# B&R Automation Studio project CombinedLinenCleanA6 (part 6)

```automation-basic
	; ###HO - 260905 - a_usCustomize[0..6]
		if(TARGETInfo_0.DataFormat = 2) then  ; motorola
			memcpy(adr(LocalCAN2Data.T3_By1),adr(LocalCOB_Typ_307.a_usCustomize[0]),1)
			memcpy(adr(LocalCAN2Data.T3_By2_By3),adr(LocalCOB_Typ_307.a_usCustomize[1]),2)
			memcpy(adr(LocalCAN2Data.T3_By4_By5),adr(LocalCOB_Typ_307.a_usCustomize[3]),2)
			memcpy(adr(LocalCAN2Data.T3_By6_By7),adr(LocalCOB_Typ_307.a_usCustomize[5]),2)
		else ; intel
			LocalCAN2Data.T3_By1 	 = LocalCOB_Typ_307.a_usCustomize[0]
			LocalCAN2Data.T3_By2_By3 = LocalCOB_Typ_307.a_usCustomize[2] + 256* LocalCOB_Typ_307.a_usCustomize[1]
			LocalCAN2Data.T3_By4_By5 = LocalCOB_Typ_307.a_usCustomize[4] + 256* LocalCOB_Typ_307.a_usCustomize[3]
			LocalCAN2Data.T3_By6_By7 = LocalCOB_Typ_307.a_usCustomize[6] + 256* LocalCOB_Typ_307.a_usCustomize[5]
		endif

    iStatus = 0
    pCAN2Data = ADR(LocalCAN2Data)
endaction ; 307

;*******action 311********action 311********action 311********action 311********action 311********
action 311: ; 311:
action 312: ; 312:
action 313: ; 313:
action 314: ; 314:
    	; ocalCOB_Typ_311 access Local_InitCAN2PV.pPVData
    	memcpy(adr(LocalCOB_Typ_311),Local_InitCAN2PV.pPVData,sizeof(LocalCOB_Typ_311))
;****ID 311****Telegram 1********ID 311****Telegram 1********ID 311****Telegram 1********ID 311****Telegram 1****
	;T1 mandatotries ->:
	; .. and sign CAN2 telegram
	LocalCAN2Data.T1_By0 = BIT_CLR(LocalCAN2Data.T1_By0, 6)
	LocalCAN2Data.T1_By0 = BIT_SET(LocalCAN2Data.T1_By0, 7)

		; bBereit
    	if LocalCOB_Typ_311.bBereit = 1 then
			LocalCAN2Data.T1_By0 = BIT_SET(LocalCAN2Data.T1_By0, 0)
		else
			LocalCAN2Data.T1_By0 = BIT_CLR(LocalCAN2Data.T1_By0, 0)
		endif
		; bBeladebereit
    	if LocalCOB_Typ_311.bBeladebereit = 1 then
			LocalCAN2Data.T1_By0 = BIT_SET(LocalCAN2Data.T1_By0, 1)
		else
			LocalCAN2Data.T1_By0 = BIT_CLR(LocalCAN2Data.T1_By0, 1)
		endif
		; bStartPresse
    	if LocalCOB_Typ_311.bStartPresse = 1 then
			LocalCAN2Data.T1_By0 = BIT_SET(LocalCAN2Data.T1_By0, 2)
		else
			LocalCAN2Data.T1_By0 = BIT_CLR(LocalCAN2Data.T1_By0, 2)
		endif
		; bUebernahmestoerungVerbETAero
    	if LocalCOB_Typ_311.bUebernahmestoerungVerbETAero = 1 then
			LocalCAN2Data.T1_By0 = BIT_SET(LocalCAN2Data.T1_By0, 3)
		else
			LocalCAN2Data.T1_By0 = BIT_CLR(LocalCAN2Data.T1_By0, 3)
		endif
		; bEntladelichtschrZentrifuge
    	if LocalCOB_Typ_311.bEntladelichtschrZentrifuge	 = 1 then
			LocalCAN2Data.T1_By0 = BIT_SET(LocalCAN2Data.T1_By0, 4)
		else
			LocalCAN2Data.T1_By0 = BIT_CLR(LocalCAN2Data.T1_By0, 4)
		endif
   ; bNotAusETVerbAero
	    if LocalCOB_Typ_311.bNotAusETVerbAero = 1 then
			LocalCAN2Data.T1_By1 = BIT_SET(LocalCAN2Data.T1_By1, 0)
		else
			LocalCAN2Data.T1_By1 = BIT_CLR(LocalCAN2Data.T1_By1, 0)
		endif
   ; bSchutzgitterOffen
	    if LocalCOB_Typ_311.bSchutzgitterOffen = 1 then
			LocalCAN2Data.T1_By1 = BIT_SET(LocalCAN2Data.T1_By1, 1)
		else
			LocalCAN2Data.T1_By1 = BIT_CLR(LocalCAN2Data.T1_By1, 1)
		endif

;****ID 311****Telegram 2********ID 311****Telegram 2********ID 311****Telegram 2********ID 311****Telegram 2****
	;T1 mandatotries ->:
	; .. and sign CAN2 telegram
	LocalCAN2Data.T2_By0 = BIT_SET(LocalCAN2Data.T2_By0, 6)
	LocalCAN2Data.T2_By0 = BIT_SET(LocalCAN2Data.T2_By0, 7)

	; ###HO - 230905 - a_usCustomize[0..6]
		if(TARGETInfo_0.DataFormat = 2) then  ; motorola
			memcpy(adr(LocalCAN2Data.T2_By1),adr(LocalCOB_Typ_311.a_usCustomize[0]),1)
			memcpy(adr(LocalCAN2Data.T2_By2_By3),adr(LocalCOB_Typ_311.a_usCustomize[1]),2)
			memcpy(adr(LocalCAN2Data.T2_By4_By5),adr(LocalCOB_Typ_311.a_usCustomize[3]),2)
			memcpy(adr(LocalCAN2Data.T2_By6_By7),adr(LocalCOB_Typ_311.a_usCustomize[5]),2)
		else ; intel
			LocalCAN2Data.T2_By1 	 = LocalCOB_Typ_311.a_usCustomize[0]
			LocalCAN2Data.T2_By2_By3 = LocalCOB_Typ_311.a_usCustomize[2] + 256* LocalCOB_Typ_311.a_usCustomize[1]
			LocalCAN2Data.T2_By4_By5 = LocalCOB_Typ_311.a_usCustomize[4] + 256* LocalCOB_Typ_311.a_usCustomize[3]
			LocalCAN2Data.T2_By6_By7 = LocalCOB_Typ_311.a_usCustomize[6] + 256* LocalCOB_Typ_311.a_usCustomize[5]
		endif

        iStatus = 0
        pCAN2Data = ADR(LocalCAN2Data)
endaction ; 311
;-----------------------------------------------------------------------------------------------------------------

;-----------------------------------------------------------------------------------------------------------------

action 316:	; 316:
    ; pLocalCOB_Typ_316 access Local_InitCAN2PV.pPVData
    memcpy(adr(LocalCOB_Typ_316),Local_InitCAN2PV.pPVData,sizeof(LocalCOB_Typ_316))
;****ID 316****Telegram 1********ID 316****Telegram 1********ID 316****Telegram 1********ID 316****Telegram 1****
	;T1 mandatotries ->:
	LocalCAN2Data.T1_By0 = BIT_CLR(LocalCAN2Data.T1_By0, 5)
	LocalCAN2Data.T1_By0 = BIT_CLR(LocalCAN2Data.T1_By0, 6)
	; .. and sign CAN2 telegram
	LocalCAN2Data.T1_By0 = BIT_SET(LocalCAN2Data.T1_By0, 7)

	; bNotAusVerbET
	   	if LocalCOB_Typ_316.bNotAusVerbET = 1 then
			LocalCAN2Data.T1_By0 = BIT_SET(LocalCAN2Data.T1_By0, 4)
		else
			LocalCAN2Data.T1_By0 = BIT_CLR(LocalCAN2Data.T1_By0, 4)
		endif
	; bBereit
    	if LocalCOB_Typ_316.bBereit = 1 then
			LocalCAN2Data.T1_By0 = BIT_SET(LocalCAN2Data.T1_By0, 0)
		else
			LocalCAN2Data.T1_By0 = BIT_CLR(LocalCAN2Data.T1_By0, 0)
		endif
	; bBeladebereit
    	if LocalCOB_Typ_316.bBeladebereit = 1 then
			LocalCAN2Data.T1_By0 = BIT_SET(LocalCAN2Data.T1_By0, 1)
		else
			LocalCAN2Data.T1_By0 = BIT_CLR(LocalCAN2Data.T1_By0, 1)
		endif
	; bUebernahmestoerungVerbET
    	if LocalCOB_Typ_316.bUebernahmestoerungVerbET = 1 then
			LocalCAN2Data.T1_By0 = BIT_SET(LocalCAN2Data.T1_By0, 3)
		else
			LocalCAN2Data.T1_By0 = BIT_CLR(LocalCAN2Data.T1_By0, 3)
		endif

	;****ID 316****Telegram 2********ID 316****Telegram 2********ID 316****Telegram 2********ID 316****Telegram 2****
	;T1 mandatotries ->:
	; .. and sign CAN2 telegram
	LocalCAN2Data.T2_By0 = BIT_SET(LocalCAN2Data.T2_By0, 5)
	LocalCAN2Data.T2_By0 = BIT_CLR(LocalCAN2Data.T2_By0, 6)
	; .. and sign CAN2 telegram
	LocalCAN2Data.T2_By0 = BIT_SET(LocalCAN2Data.T2_By0, 7)

	; ###HO - 230905 - a_usCustomize[0..6]
	if(TARGETInfo_0.DataFormat = 2) then  ; motorola
		memcpy(adr(LocalCAN2Data.T2_By1),adr(LocalCOB_Typ_316.a_usCustomize[0]),1)
		memcpy(adr(LocalCAN2Data.T2_By2_By3),adr(LocalCOB_Typ_316.a_usCustomize[1]),2)
		memcpy(adr(LocalCAN2Data.T2_By4_By5),adr(LocalCOB_Typ_316.a_usCustomize[3]),2)
		memcpy(adr(LocalCAN2Data.T2_By6_By7),adr(LocalCOB_Typ_316.a_usCustomize[5]),2)
	else ; intel
		LocalCAN2Data.T2_By1 	 = LocalCOB_Typ_316.a_usCustomize[0]
		LocalCAN2Data.T2_By2_By3 = LocalCOB_Typ_316.a_usCustomize[2] + 256* LocalCOB_Typ_316.a_usCustomize[1]
		LocalCAN2Data.T2_By4_By5 = LocalCOB_Typ_316.a_usCustomize[4] + 256* LocalCOB_Typ_316.a_usCustomize[3]
		LocalCAN2Data.T2_By6_By7 = LocalCOB_Typ_316.a_usCustomize[6] + 256* LocalCOB_Typ_316.a_usCustomize[5]
	endif

    iStatus = 0
    pCAN2Data = ADR(LocalCAN2Data)

endaction ; 316

;*******action 317********action 317********action 317********action 317********action 317********
action 317: ; 317:
    	; pLocalCOB_Typ_317 access Local_InitCAN2PV.pPVData
    	memcpy(adr(LocalCOB_Typ_317),Local_InitCAN2PV.pPVData,sizeof(LocalCOB_Typ_317))

;****ID 317****Telegram 1********ID 317****Telegram 1********ID 317****Telegram 1********ID 317****Telegram 1****
	;T1 mandatotries ->:
	LocalCAN2Data.T1_By0 = BIT_CLR(LocalCAN2Data.T1_By0, 6)
	; .. and sign CAN2 telegram
	LocalCAN2Data.T1_By0 = BIT_SET(LocalCAN2Data.T1_By0, 7)

;	bBereit
    	if LocalCOB_Typ_317.bBereit = 1 then
			LocalCAN2Data.T1_By0 = BIT_SET(LocalCAN2Data.T1_By0, 0)
		else
			LocalCAN2Data.T1_By0 = BIT_CLR(LocalCAN2Data.T1_By0, 0)
		endif
;	bBeladebereit
    	if LocalCOB_Typ_317.bBeladebereit = 1 then
			LocalCAN2Data.T1_By0 = BIT_SET(LocalCAN2Data.T1_By0, 1)
		else
			LocalCAN2Data.T1_By0 = BIT_CLR(LocalCAN2Data.T1_By0, 1)
		endif
;	bBeladeunterbrechung
    	if LocalCOB_Typ_317.bBeladeunterbrechung = 1 then
			LocalCAN2Data.T1_By0 = BIT_SET(LocalCAN2Data.T1_By0, 2)
		else
			LocalCAN2Data.T1_By0 = BIT_CLR(LocalCAN2Data.T1_By0, 2)
		endif
;	bUebernahmestoerung
    	if LocalCOB_Typ_317.bUebernahmestoerung = 1 then
			LocalCAN2Data.T1_By0 = BIT_SET(LocalCAN2Data.T1_By0, 3)
		else
			LocalCAN2Data.T1_By0 = BIT_CLR(LocalCAN2Data.T1_By0, 3)
		endif
;	bQuittierungKundenwechsel
    	if LocalCOB_Typ_317.bQuittierungKundenwechsel = 1 then
			LocalCAN2Data.T1_By0 = BIT_SET(LocalCAN2Data.T1_By0, 4)
		else
			LocalCAN2Data.T1_By0 = BIT_CLR(LocalCAN2Data.T1_By0, 4)
		endif
;	bNotAusAero
    	if LocalCOB_Typ_317.bNotAusAero = 1 then
			LocalCAN2Data.T1_By0 = BIT_SET(LocalCAN2Data.T1_By0, 5)
		else
			LocalCAN2Data.T1_By0 = BIT_CLR(LocalCAN2Data.T1_By0, 5)
		endif
;****ID 317****Telegram 2********ID 317****Telegram 2********ID 317****Telegram 2********ID 317****Telegram 2****
	; always set telegram number "01"..
	LocalCAN2Data.T2_By0 = BIT_SET(LocalCAN2Data.T2_By0, 6)
	; .. and sign CAN2 telegram
	LocalCAN2Data.T2_By0 = BIT_SET(LocalCAN2Data.T2_By0, 7)

   	; ###HO - 260905 - a_usCustomize[0..6]
		if(TARGETInfo_0.DataFormat = 2) then  ; motorola
			memcpy(adr(LocalCAN2Data.T2_By1),adr(LocalCOB_Typ_317.a_usCustomize[0]),1)
			memcpy(adr(LocalCAN2Data.T2_By2_By3),adr(LocalCOB_Typ_317.a_usCustomize[1]),2)
			memcpy(adr(LocalCAN2Data.T2_By4_By5),adr(LocalCOB_Typ_317.a_usCustomize[3]),2)
			memcpy(adr(LocalCAN2Data.T2_By6_By7),adr(LocalCOB_Typ_317.a_usCustomize[5]),2)
		else ; intel
			LocalCAN2Data.T2_By1	 = LocalCOB_Typ_317.a_usCustomize[0]
			LocalCAN2Data.T2_By2_By3 = LocalCOB_Typ_317.a_usCustomize[2] + 256* LocalCOB_Typ_317.a_usCustomize[1]
			LocalCAN2Data.T2_By4_By5 = LocalCOB_Typ_317.a_usCustomize[4] + 256* LocalCOB_Typ_317.a_usCustomize[3]
			LocalCAN2Data.T2_By6_By7 = LocalCOB_Typ_317.a_usCustomize[6] + 256* LocalCOB_Typ_317.a_usCustomize[5]
		endif

  	iStatus = 0
    pCAN2Data = ADR(LocalCAN2Data)
endaction ; 317

;*******action 351********action 351********action 351********action 351********action 351********
action 351: ; 351:
    	; pLocalCOB_Typ_351 access Local_InitCAN2PV.pPVData
    	memcpy(adr(LocalCOB_Typ_351),Local_InitCAN2PV.pPVData,sizeof(LocalCOB_Typ_351))

;****ID 351****Telegram 1********ID 351****Telegram 1********ID 351****Telegram 1********ID 351****Telegram 1****
		;T1 mandatotries ->:
		LocalCAN2Data.T1_By0 = BIT_CLR(LocalCAN2Data.T1_By0, 5)
		LocalCAN2Data.T1_By0 = BIT_CLR(LocalCAN2Data.T1_By0, 6)
		; .. and sign CAN2 telegram
		LocalCAN2Data.T1_By0 = BIT_SET(LocalCAN2Data.T1_By0, 7)

;	bBereit
    	if LocalCOB_Typ_351.bBereit = 1 then
			LocalCAN2Data.T1_By0 = BIT_SET(LocalCAN2Data.T1_By0, 0)
		else
				LocalCAN2Data.T1_By0 = BIT_CLR(LocalCAN2Data.T1_By0, 0)
		endif
;	bAktPosFehler
    	if LocalCOB_Typ_351.bAktPosFehler = 1 then
			LocalCAN2Data.T1_By0 = BIT_SET(LocalCAN2Data.T1_By0, 1)
		else
			LocalCAN2Data.T1_By0 = BIT_CLR(LocalCAN2Data.T1_By0, 1)
		endif
;	bIdxPostenindex_x - 110107
    	if LocalCOB_Typ_351.bIdxPostenspeicher_1 = 1 then
			LocalCAN2Data.T1_By0 = BIT_SET(LocalCAN2Data.T1_By0, 2)
		else
			LocalCAN2Data.T1_By0 = BIT_CLR(LocalCAN2Data.T1_By0, 2)
		endif
		if LocalCOB_Typ_351.bIdxPostenspeicher_2 = 1 then
			LocalCAN2Data.T1_By0 = BIT_SET(LocalCAN2Data.T1_By0, 3)
		else
			LocalCAN2Data.T1_By0 = BIT_CLR(LocalCAN2Data.T1_By0, 3)
		endif
		if LocalCOB_Typ_351.bIdxPostenspeicher_4 = 1 then
			LocalCAN2Data.T1_By0 = BIT_SET(LocalCAN2Data.T1_By0, 4)
		else
			LocalCAN2Data.T1_By0 = BIT_CLR(LocalCAN2Data.T1_By0, 4)
		endif
;	usAktPos
		LocalCAN2Data.T1_By1	= LocalCOB_Typ_351.usAktPos
;	udPostennummer				8-11
			udShr16 = shr(LocalCOB_Typ_351.udPostennummer,16)
    	LocalCAN2Data.T1_By2_By3	= UINT(udShr16)							; take UPPERBytes ..
    	LocalCAN2Data.T1_By4_By5	= UINT(LocalCOB_Typ_351.udPostennummer)	; take LOWER byte..
;	uiGewicht					16-17
		LocalCAN2Data.T1_By6_By7	= LocalCOB_Typ_351.uiGewicht

;****ID 351****Telegram 2********ID 351****Telegram 2********ID 351****Telegram 2********ID 351****Telegram 2****
		; always set telegram number "01"..
		LocalCAN2Data.T2_By0 = BIT_CLR(LocalCAN2Data.T2_By0, 5)
		LocalCAN2Data.T2_By0 = BIT_SET(LocalCAN2Data.T2_By0, 6)
		; .. and sign CAN2 telegram
		LocalCAN2Data.T2_By0 = BIT_SET(LocalCAN2Data.T2_By0, 7)

		; bProgrammOderKategorie
    	if LocalCOB_Typ_351.bProgrammOderKategorie = 1 then
			LocalCAN2Data.T2_By0 = BIT_SET(LocalCAN2Data.T2_By0, 0)
		else
			LocalCAN2Data.T2_By0 = BIT_CLR(LocalCAN2Data.T2_By0, 0)
		endif
		;	bNotAusAero
    	if LocalCOB_Typ_351.bNotAusAero = 1 then
			LocalCAN2Data.T2_By0 = BIT_SET(LocalCAN2Data.T2_By0, 1)
		else
			LocalCAN2Data.T2_By0 = BIT_CLR(LocalCAN2Data.T2_By0, 1)
		endif
;		uiProgrammKategorie
		LocalCAN2Data.T2_By2_By3	= LocalCOB_Typ_351.uiProgrammKategorie
    	; udKundennummer
	   	 	udShr16 = shr(LocalCOB_Typ_351.udKundennummer,16)
    	LocalCAN2Data.T2_By4_By5	= UINT(udShr16)							; take UPPERBytes ..
    	LocalCAN2Data.T2_By6_By7	= UINT(LocalCOB_Typ_351.udKundennummer)	; take LOWER bytes..

;****ID 351****Telegram 3********ID 351****Telegram 3********ID 351****Telegram 3********ID 351****Telegram 3****
		; always set telegram number "01"..
		LocalCAN2Data.T3_By0 = BIT_SET(LocalCAN2Data.T3_By0, 5)
		LocalCAN2Data.T3_By0 = BIT_CLR(LocalCAN2Data.T3_By0, 6)
		; .. and sign CAN2 telegram
		LocalCAN2Data.T3_By0 = BIT_SET(LocalCAN2Data.T3_By0, 7)
;	bAktPosGesperrt
    	if LocalCOB_Typ_351.bAktPosGesperrt = 1 then
			LocalCAN2Data.T3_By0 = BIT_SET(LocalCAN2Data.T3_By0, 0)
		else
			LocalCAN2Data.T3_By0 = BIT_CLR(LocalCAN2Data.T3_By0, 0)
		endif
;	bAktPosWarnung
    	if LocalCOB_Typ_351.bAktPosWarnung = 1 then
			LocalCAN2Data.T3_By0 = BIT_SET(LocalCAN2Data.T3_By0, 1)
		else
			LocalCAN2Data.T3_By0 = BIT_CLR(LocalCAN2Data.T3_By0, 1)
		endif
	; ###HO - 110107 - a_usCustomize[0..6]
		if(TARGETInfo_0.DataFormat = 2) then  ; motorola
			memcpy(adr(LocalCAN2Data.T3_By1),adr(LocalCOB_Typ_351.a_usCustomize[0]),1)
			memcpy(adr(LocalCAN2Data.T3_By2_By3),adr(LocalCOB_Typ_351.a_usCustomize[1]),2)
			memcpy(adr(LocalCAN2Data.T3_By4_By5),adr(LocalCOB_Typ_351.a_usCustomize[3]),2)
			memcpy(adr(LocalCAN2Data.T3_By6_By7),adr(LocalCOB_Typ_351.a_usCustomize[5]),2)
		else ; intel
			LocalCAN2Data.T3_By1 	 = LocalCOB_Typ_351.a_usCustomize[0]
			LocalCAN2Data.T3_By2_By3 = LocalCOB_Typ_351.a_usCustomize[2] + 256* LocalCOB_Typ_351.a_usCustomize[1]
			LocalCAN2Data.T3_By4_By5 = LocalCOB_Typ_351.a_usCustomize[4] + 256* LocalCOB_Typ_351.a_usCustomize[3]
			LocalCAN2Data.T3_By6_By7 = LocalCOB_Typ_351.a_usCustomize[6] + 256* LocalCOB_Typ_351.a_usCustomize[5]
		endif

    iStatus = 0
    pCAN2Data = ADR(LocalCAN2Data)
endaction 	; 351

;*******action 352********action 352********action 352********action 352********action 352********
action 352: ; 352:
    	; pLocalCOB_Typ_352 access Local_InitCAN2PV.pPVData
    	memcpy(adr(LocalCOB_Typ_352),Local_InitCAN2PV.pPVData,sizeof(LocalCOB_Typ_352))

;****ID 352****Telegram 1********ID 352****Telegram 1********ID 352****Telegram 1********ID 352****Telegram 1****
		;T1 mandatotries ->:
		LocalCAN2Data.T1_By0 = BIT_CLR(LocalCAN2Data.T1_By0, 5)
		LocalCAN2Data.T1_By0 = BIT_CLR(LocalCAN2Data.T1_By0, 6)
		; .. and sign CAN2 telegram
		LocalCAN2Data.T1_By0 = BIT_SET(LocalCAN2Data.T1_By0, 7)

;	bBereit
    	if LocalCOB_Typ_352.bBereit = 1 then
			LocalCAN2Data.T1_By0 = BIT_SET(LocalCAN2Data.T1_By0, 0)
		else
				LocalCAN2Data.T1_By0 = BIT_CLR(LocalCAN2Data.T1_By0, 0)
		endif
;	bAktPosFehler
    	if LocalCOB_Typ_352.bAktPosFehler = 1 then
			LocalCAN2Data.T1_By0 = BIT_SET(LocalCAN2Data.T1_By0, 1)
		else
			LocalCAN2Data.T1_By0 = BIT_CLR(LocalCAN2Data.T1_By0, 1)
		endif
;	bIdxPostenindex_x - 110107
    	if LocalCOB_Typ_352.bIdxPostenspeicher_1 = 1 then
			LocalCAN2Data.T1_By0 = BIT_SET(LocalCAN2Data.T1_By0, 2)
		else
			LocalCAN2Data.T1_By0 = BIT_CLR(LocalCAN2Data.T1_By0, 2)
		endif
		if LocalCOB_Typ_352.bIdxPostenspeicher_2 = 1 then
			LocalCAN2Data.T1_By0 = BIT_SET(LocalCAN2Data.T1_By0, 3)
		else
			LocalCAN2Data.T1_By0 = BIT_CLR(LocalCAN2Data.T1_By0, 3)
		endif
		if LocalCOB_Typ_352.bIdxPostenspeicher_4 = 1 then
			LocalCAN2Data.T1_By0 = BIT_SET(LocalCAN2Data.T1_By0, 4)
		else
			LocalCAN2Data.T1_By0 = BIT_CLR(LocalCAN2Data.T1_By0, 4)
		endif
;	usAktPos
		LocalCAN2Data.T1_By1	= LocalCOB_Typ_352.usAktPos
;	udPostennummer				8-11
			udShr16 = shr(LocalCOB_Typ_352.udPostennummer,16)
    	LocalCAN2Data.T1_By2_By3	= UINT(udShr16)							; take UPPERBytes ..
    	LocalCAN2Data.T1_By4_By5	= UINT(LocalCOB_Typ_352.udPostennummer)	; take LOWER byte..
;	uiGewicht					16-17
		LocalCAN2Data.T1_By6_By7	= LocalCOB_Typ_352.uiGewicht

;****ID 352****Telegram 2********ID 352****Telegram 2********ID 352****Telegram 2********ID 352****Telegram 2****
		; always set telegram number "01"..
		LocalCAN2Data.T2_By0 = BIT_CLR(LocalCAN2Data.T2_By0, 5)
		LocalCAN2Data.T2_By0 = BIT_SET(LocalCAN2Data.T2_By0, 6)
		; .. and sign CAN2 telegram
		LocalCAN2Data.T2_By0 = BIT_SET(LocalCAN2Data.T2_By0, 7)

		; bProgrammOderKategorie
    	if LocalCOB_Typ_352.bProgrammOderKategorie = 1 then
			LocalCAN2Data.T2_By0 = BIT_SET(LocalCAN2Data.T2_By0, 0)
		else
			LocalCAN2Data.T2_By0 = BIT_CLR(LocalCAN2Data.T2_By0, 0)
		endif
		;	bNotAusAero
    	if LocalCOB_Typ_352.bNotAusAero = 1 then
			LocalCAN2Data.T2_By0 = BIT_SET(LocalCAN2Data.T2_By0, 1)
		else
			LocalCAN2Data.T2_By0 = BIT_CLR(LocalCAN2Data.T2_By0, 1)
		endif
;		uiProgrammKategorie
		LocalCAN2Data.T2_By2_By3	= LocalCOB_Typ_352.uiProgrammKategorie
    	; udKundennummer
	   	 	udShr16 = shr(LocalCOB_Typ_352.udKundennummer,16)
    	LocalCAN2Data.T2_By4_By5	= UINT(udShr16)							; take UPPERBytes ..
    	LocalCAN2Data.T2_By6_By7	= UINT(LocalCOB_Typ_352.udKundennummer)	; take LOWER bytes..

;****ID 352****Telegram 3********ID 352****Telegram 3********ID 352****Telegram 3********ID 352****Telegram 3****
		; always set telegram number "01"..
		LocalCAN2Data.T3_By0 = BIT_SET(LocalCAN2Data.T3_By0, 5)
		LocalCAN2Data.T3_By0 = BIT_CLR(LocalCAN2Data.T3_By0, 6)
		; .. and sign CAN2 telegram
		LocalCAN2Data.T3_By0 = BIT_SET(LocalCAN2Data.T3_By0, 7)
;	bAktPosGesperrt
    	if LocalCOB_Typ_352.bAktPosGesperrt = 1 then
			LocalCAN2Data.T3_By0 = BIT_SET(LocalCAN2Data.T3_By0, 0)
		else
			LocalCAN2Data.T3_By0 = BIT_CLR(LocalCAN2Data.T3_By0, 0)
		endif
;	bAktPosWarnung
    	if LocalCOB_Typ_352.bAktPosWarnung = 1 then
			LocalCAN2Data.T3_By0 = BIT_SET(LocalCAN2Data.T3_By0, 1)
		else
			LocalCAN2Data.T3_By0 = BIT_CLR(LocalCAN2Data.T3_By0, 1)
		endif
	; ###HO - 110107 - a_usCustomize[0..6]
		if(TARGETInfo_0.DataFormat = 2) then  ; motorola
			memcpy(adr(LocalCAN2Data.T3_By1),adr(LocalCOB_Typ_352.a_usCustomize[0]),1)
			memcpy(adr(LocalCAN2Data.T3_By2_By3),adr(LocalCOB_Typ_352.a_usCustomize[1]),2)
			memcpy(adr(LocalCAN2Data.T3_By4_By5),adr(LocalCOB_Typ_352.a_usCustomize[3]),2)
			memcpy(adr(LocalCAN2Data.T3_By6_By7),adr(LocalCOB_Typ_352.a_usCustomize[5]),2)
		else ; intel
			LocalCAN2Data.T3_By1 	 = LocalCOB_Typ_352.a_usCustomize[0]
			LocalCAN2Data.T3_By2_By3 = LocalCOB_Typ_352.a_usCustomize[2] + 256* LocalCOB_Typ_352.a_usCustomize[1]
			LocalCAN2Data.T3_By4_By5 = LocalCOB_Typ_352.a_usCustomize[4] + 256* LocalCOB_Typ_352.a_usCustomize[3]
			LocalCAN2Data.T3_By6_By7 = LocalCOB_Typ_352.a_usCustomize[6] + 256* LocalCOB_Typ_352.a_usCustomize[5]
		endif

    iStatus = 0
    pCAN2Data = ADR(LocalCAN2Data)
endaction 	; 352

;*******action 353********action 353********action 353********action 353********action 353********
action 353: ; 353:
    	; pLocalCOB_Typ_353 access Local_InitCAN2PV.pPVData
    	memcpy(adr(LocalCOB_Typ_353),Local_InitCAN2PV.pPVData,sizeof(LocalCOB_Typ_353))

;****ID 353****Telegram 1********ID 353****Telegram 1********ID 353****Telegram 1********ID 353****Telegram 1****
		;T1 mandatotries ->:
		LocalCAN2Data.T1_By0 = BIT_CLR(LocalCAN2Data.T1_By0, 5)
		LocalCAN2Data.T1_By0 = BIT_CLR(LocalCAN2Data.T1_By0, 6)
		; .. and sign CAN2 telegram
		LocalCAN2Data.T1_By0 = BIT_SET(LocalCAN2Data.T1_By0, 7)

;	bBereit
    	if LocalCOB_Typ_353.bBereit = 1 then
			LocalCAN2Data.T1_By0 = BIT_SET(LocalCAN2Data.T1_By0, 0)
		else
				LocalCAN2Data.T1_By0 = BIT_CLR(LocalCAN2Data.T1_By0, 0)
		endif
;	bAktPosFehler
    	if LocalCOB_Typ_353.bAktPosFehler = 1 then
			LocalCAN2Data.T1_By0 = BIT_SET(LocalCAN2Data.T1_By0, 1)
		else
			LocalCAN2Data.T1_By0 = BIT_CLR(LocalCAN2Data.T1_By0, 1)
		endif
;	bIdxPostenindex_x - 110107
    	if LocalCOB_Typ_353.bIdxPostenspeicher_1 = 1 then

			LocalCAN2Data.T1_By0 = BIT_SET(LocalCAN2Data.T1_By0, 2)
		else
			LocalCAN2Data.T1_By0 = BIT_CLR(LocalCAN2Data.T1_By0, 2)
		endif
		if LocalCOB_Typ_353.bIdxPostenspeicher_2 = 1 then
			LocalCAN2Data.T1_By0 = BIT_SET(LocalCAN2Data.T1_By0, 3)
		else
			LocalCAN2Data.T1_By0 = BIT_CLR(LocalCAN2Data.T1_By0, 3)
		endif
		if LocalCOB_Typ_353.bIdxPostenspeicher_4 = 1 then
			LocalCAN2Data.T1_By0 = BIT_SET(LocalCAN2Data.T1_By0, 4)
		else
			LocalCAN2Data.T1_By0 = BIT_CLR(LocalCAN2Data.T1_By0, 4)
		endif
;	usAktPos
		LocalCAN2Data.T1_By1	= LocalCOB_Typ_353.usAktPos
;	udPostennummer				8-11
			udShr16 = shr(LocalCOB_Typ_353.udPostennummer,16)
    	LocalCAN2Data.T1_By2_By3	= UINT(udShr16)							; take UPPERBytes ..
    	LocalCAN2Data.T1_By4_By5	= UINT(LocalCOB_Typ_353.udPostennummer)	; take LOWER byte..
;	uiGewicht					16-17
		LocalCAN2Data.T1_By6_By7	= LocalCOB_Typ_353.uiGewicht

;****ID 353****Telegram 2********ID 353****Telegram 2********ID 353****Telegram 2********ID 353****Telegram 2****
		; always set telegram number "01"..
		LocalCAN2Data.T2_By0 = BIT_CLR(LocalCAN2Data.T2_By0, 5)
		LocalCAN2Data.T2_By0 = BIT_SET(LocalCAN2Data.T2_By0, 6)
		; .. and sign CAN2 telegram
		LocalCAN2Data.T2_By0 = BIT_SET(LocalCAN2Data.T2_By0, 7)

		; bProgrammOderKategorie
    	if LocalCOB_Typ_353.bProgrammOderKategorie = 1 then
			LocalCAN2Data.T2_By0 = BIT_SET(LocalCAN2Data.T2_By0, 0)
		else
			LocalCAN2Data.T2_By0 = BIT_CLR(LocalCAN2Data.T2_By0, 0)
		endif
		;	bNotAusAero
    	if LocalCOB_Typ_353.bNotAusAero = 1 then
			LocalCAN2Data.T2_By0 = BIT_SET(LocalCAN2Data.T2_By0, 1)
		else
			LocalCAN2Data.T2_By0 = BIT_CLR(LocalCAN2Data.T2_By0, 1)
		endif
;		uiProgrammKategorie
		LocalCAN2Data.T2_By2_By3	= LocalCOB_Typ_353.uiProgrammKategorie
    	; udKundennummer
	   	 	udShr16 = shr(LocalCOB_Typ_353.udKundennummer,16)
    	LocalCAN2Data.T2_By4_By5	= UINT(udShr16)							; take UPPERBytes ..
    	LocalCAN2Data.T2_By6_By7	= UINT(LocalCOB_Typ_353.udKundennummer)	; take LOWER bytes..

;****ID 353****Telegram 3********ID 353****Telegram 3********ID 353****Telegram 3********ID 353****Telegram 3****
		; always set telegram number "01"..
		LocalCAN2Data.T3_By0 = BIT_SET(LocalCAN2Data.T3_By0, 5)
		LocalCAN2Data.T3_By0 = BIT_CLR(LocalCAN2Data.T3_By0, 6)
		; .. and sign CAN2 telegram
		LocalCAN2Data.T3_By0 = BIT_SET(LocalCAN2Data.T3_By0, 7)
;	bAktPosGesperrt
    	if LocalCOB_Typ_353.bAktPosGesperrt = 1 then
			LocalCAN2Data.T3_By0 = BIT_SET(LocalCAN2Data.T3_By0, 0)
		else
			LocalCAN2Data.T3_By0 = BIT_CLR(LocalCAN2Data.T3_By0, 0)
		endif
;	bAktPosWarnung
    	if LocalCOB_Typ_353.bAktPosWarnung = 1 then
			LocalCAN2Data.T3_By0 = BIT_SET(LocalCAN2Data.T3_By0, 1)
		else
			LocalCAN2Data.T3_By0 = BIT_CLR(LocalCAN2Data.T3_By0, 1)
		endif
	; ###HO - 110107 - a_usCustomize[0..6]
		if(TARGETInfo_0.DataFormat = 2) then  ; motorola
			memcpy(adr(LocalCAN2Data.T3_By1),adr(LocalCOB_Typ_353.a_usCustomize[0]),1)
			memcpy(adr(LocalCAN2Data.T3_By2_By3),adr(LocalCOB_Typ_353.a_usCustomize[1]),2)
			memcpy(adr(LocalCAN2Data.T3_By4_By5),adr(LocalCOB_Typ_353.a_usCustomize[3]),2)
			memcpy(adr(LocalCAN2Data.T3_By6_By7),adr(LocalCOB_Typ_353.a_usCustomize[5]),2)
		else ; intel
			LocalCAN2Data.T3_By1 	 = LocalCOB_Typ_353.a_usCustomize[0]
			LocalCAN2Data.T3_By2_By3 = LocalCOB_Typ_353.a_usCustomize[2] + 256* LocalCOB_Typ_353.a_usCustomize[1]
			LocalCAN2Data.T3_By4_By5 = LocalCOB_Typ_353.a_usCustomize[4] + 256* LocalCOB_Typ_353.a_usCustomize[3]
			LocalCAN2Data.T3_By6_By7 = LocalCOB_Typ_353.a_usCustomize[6] + 256* LocalCOB_Typ_353.a_usCustomize[5]
		endif

    iStatus = 0
    pCAN2Data = ADR(LocalCAN2Data)
endaction 	; 353

;*******action 354********action 354********action 354********action 354********action 354********
action 354: ; 354:
    	; pLocalCOB_Typ_354 access Local_InitCAN2PV.pPVData
    	memcpy(adr(LocalCOB_Typ_354),Local_InitCAN2PV.pPVData,sizeof(LocalCOB_Typ_354))

;****ID 354****Telegram 1********ID 354****Telegram 1********ID 354****Telegram 1********ID 354****Telegram 1****
		;T1 mandatotries ->:
		LocalCAN2Data.T1_By0 = BIT_CLR(LocalCAN2Data.T1_By0, 5)
		LocalCAN2Data.T1_By0 = BIT_CLR(LocalCAN2Data.T1_By0, 6)
		; .. and sign CAN2 telegram
		LocalCAN2Data.T1_By0 = BIT_SET(LocalCAN2Data.T1_By0, 7)

;	bBereit
    	if LocalCOB_Typ_354.bBereit = 1 then
			LocalCAN2Data.T1_By0 = BIT_SET(LocalCAN2Data.T1_By0, 0)
		else
				LocalCAN2Data.T1_By0 = BIT_CLR(LocalCAN2Data.T1_By0, 0)
		endif
;	bAktPosFehler
    	if LocalCOB_Typ_354.bAktPosFehler = 1 then
			LocalCAN2Data.T1_By0 = BIT_SET(LocalCAN2Data.T1_By0, 1)
		else
			LocalCAN2Data.T1_By0 = BIT_CLR(LocalCAN2Data.T1_By0, 1)
		endif
;	bIdxPostenindex_x - 110107
    	if LocalCOB_Typ_354.bIdxPostenspeicher_1 = 1 then
			LocalCAN2Data.T1_By0 = BIT_SET(LocalCAN2Data.T1_By0, 2)
		else
			LocalCAN2Data.T1_By0 = BIT_CLR(LocalCAN2Data.T1_By0, 2)
		endif
		if LocalCOB_Typ_354.bIdxPostenspeicher_2 = 1 then
			LocalCAN2Data.T1_By0 = BIT_SET(LocalCAN2Data.T1_By0, 3)
		else
			LocalCAN2Data.T1_By0 = BIT_CLR(LocalCAN2Data.T1_By0, 3)
		endif
		if LocalCOB_Typ_354.bIdxPostenspeicher_4 = 1 then
			LocalCAN2Data.T1_By0 = BIT_SET(LocalCAN2Data.T1_By0, 4)
		else
			LocalCAN2Data.T1_By0 = BIT_CLR(LocalCAN2Data.T1_By0, 4)
		endif
;	usAktPos
		LocalCAN2Data.T1_By1	= LocalCOB_Typ_354.usAktPos
;	udPostennummer				8-11
			udShr16 = shr(LocalCOB_Typ_354.udPostennummer,16)
    	LocalCAN2Data.T1_By2_By3	= UINT(udShr16)							; take UPPERBytes ..
    	LocalCAN2Data.T1_By4_By5	= UINT(LocalCOB_Typ_354.udPostennummer)	; take LOWER byte..
;	uiGewicht					16-17
		LocalCAN2Data.T1_By6_By7	= LocalCOB_Typ_354.uiGewicht

;****ID 354****Telegram 2********ID 354****Telegram 2********ID 354****Telegram 2********ID 354****Telegram 2****
		; always set telegram number "01"..
		LocalCAN2Data.T2_By0 = BIT_CLR(LocalCAN2Data.T2_By0, 5)
		LocalCAN2Data.T2_By0 = BIT_SET(LocalCAN2Data.T2_By0, 6)
		; .. and sign CAN2 telegram
		LocalCAN2Data.T2_By0 = BIT_SET(LocalCAN2Data.T2_By0, 7)

		; bProgrammOderKategorie
    	if LocalCOB_Typ_354.bProgrammOderKategorie = 1 then
			LocalCAN2Data.T2_By0 = BIT_SET(LocalCAN2Data.T2_By0, 0)
		else
			LocalCAN2Data.T2_By0 = BIT_CLR(LocalCAN2Data.T2_By0, 0)
		endif
		;	bNotAusAero
    	if LocalCOB_Typ_354.bNotAusAero = 1 then
			LocalCAN2Data.T2_By0 = BIT_SET(LocalCAN2Data.T2_By0, 1)
		else
			LocalCAN2Data.T2_By0 = BIT_CLR(LocalCAN2Data.T2_By0, 1)
		endif
;		uiProgrammKategorie
		LocalCAN2Data.T2_By2_By3	= LocalCOB_Typ_354.uiProgrammKategorie
    	; udKundennummer
	   	 	udShr16 = shr(LocalCOB_Typ_354.udKundennummer,16)
    	LocalCAN2Data.T2_By4_By5	= UINT(udShr16)							; take UPPERBytes ..
    	LocalCAN2Data.T2_By6_By7	= UINT(LocalCOB_Typ_354.udKundennummer)	; take LOWER bytes..

;****ID 354****Telegram 3********ID 354****Telegram 3********ID 354****Telegram 3********ID 354****Telegram 3****
		; always set telegram number "01"..
		LocalCAN2Data.T3_By0 = BIT_SET(LocalCAN2Data.T3_By0, 5)
		LocalCAN2Data.T3_By0 = BIT_CLR(LocalCAN2Data.T3_By0, 6)
		; .. and sign CAN2 telegram
		LocalCAN2Data.T3_By0 = BIT_SET(LocalCAN2Data.T3_By0, 7)
;	bAktPosGesperrt
    	if LocalCOB_Typ_354.bAktPosGesperrt = 1 then
			LocalCAN2Data.T3_By0 = BIT_SET(LocalCAN2Data.T3_By0, 0)
		else
			LocalCAN2Data.T3_By0 = BIT_CLR(LocalCAN2Data.T3_By0, 0)
		endif
;	bAktPosWarnung
    	if LocalCOB_Typ_354.bAktPosWarnung = 1 then
			LocalCAN2Data.T3_By0 = BIT_SET(LocalCAN2Data.T3_By0, 1)
		else
			LocalCAN2Data.T3_By0 = BIT_CLR(LocalCAN2Data.T3_By0, 1)
		endif
	; ###HO - 110107 - a_usCustomize[0..6]
		if(TARGETInfo_0.DataFormat = 2) then  ; motorola
			memcpy(adr(LocalCAN2Data.T3_By1),adr(LocalCOB_Typ_354.a_usCustomize[0]),1)
			memcpy(adr(LocalCAN2Data.T3_By2_By3),adr(LocalCOB_Typ_354.a_usCustomize[1]),2)
			memcpy(adr(LocalCAN2Data.T3_By4_By5),adr(LocalCOB_Typ_354.a_usCustomize[3]),2)
			memcpy(adr(LocalCAN2Data.T3_By6_By7),adr(LocalCOB_Typ_354.a_usCustomize[5]),2)
		else ; intel
			LocalCAN2Data.T3_By1 	 = LocalCOB_Typ_354.a_usCustomize[0]
			LocalCAN2Data.T3_By2_By3 = LocalCOB_Typ_354.a_usCustomize[2] + 256* LocalCOB_Typ_354.a_usCustomize[1]
			LocalCAN2Data.T3_By4_By5 = LocalCOB_Typ_354.a_usCustomize[4] + 256* LocalCOB_Typ_354.a_usCustomize[3]
			LocalCAN2Data.T3_By6_By7 = LocalCOB_Typ_354.a_usCustomize[6] + 256* LocalCOB_Typ_354.a_usCustomize[5]
		endif

    iStatus = 0
    pCAN2Data = ADR(LocalCAN2Data)
endaction 	; 354
;;;
;*******action 361..369********action 361..369********action 361..369********action 361..369********action 361..369********
action 361..369: ; 361..369:
    	; pLocalCOB_Typ_361bis369 access Local_InitCAN2PV.pPVData
    	memcpy(adr(LocalCOB_Typ_361bis369),Local_InitCAN2PV.pPVData,sizeof(LocalCOB_Typ_361bis369))

;****ID 361..369****Telegram 1********ID 361..369****Telegram 1********ID 361..369****Telegram 1********ID 361..369****Telegram 1****
	;T1 mandatotries ->:
		LocalCAN2Data.T1_By0 = BIT_CLR(LocalCAN2Data.T1_By0, 5)
		LocalCAN2Data.T1_By0 = BIT_CLR(LocalCAN2Data.T1_By0, 6)
	; .. and sign CAN2 telegram
		LocalCAN2Data.T1_By0 = BIT_SET(LocalCAN2Data.T1_By0, 7)
	; bBereit
    	if LocalCOB_Typ_361bis369.bBereit = 1 then
			LocalCAN2Data.T1_By0 = BIT_SET(LocalCAN2Data.T1_By0, 0)
		else
			LocalCAN2Data.T1_By0 = BIT_CLR(LocalCAN2Data.T1_By0, 0)
		endif
	; usStation
		LocalCAN2Data.T1_By1	= LocalCOB_Typ_361bis369.usStation
	; udPostennummer
			udShr16 = shr(LocalCOB_Typ_361bis369.udPostennummer,16)
	   	LocalCAN2Data.T1_By2_By3	= UINT(udShr16)								; take UPPERBytes ..
	   	LocalCAN2Data.T1_By4_By5	= UINT(LocalCOB_Typ_361bis369.udPostennummer)	; take LOWER byte..
	; uiGewicht
		LocalCAN2Data.T1_By6_By7	= LocalCOB_Typ_361bis369.uiGewicht

;****ID 361..369****Telegram 2********ID 361..369****Telegram 2********ID 361..369****Telegram 2********ID 361..369****Telegram 2****
		; always set telegram number "01"..
		LocalCAN2Data.T2_By0 = BIT_SET(LocalCAN2Data.T2_By0, 5)
		LocalCAN2Data.T2_By0 = BIT_CLR(LocalCAN2Data.T2_By0, 6)
		; .. and sign CAN2 telegram
		LocalCAN2Data.T2_By0 = BIT_SET(LocalCAN2Data.T2_By0, 7)

	; bProgrammOderKategorie
    	if LocalCOB_Typ_361bis369.bProgrammOderKategorie = 1 then
			LocalCAN2Data.T2_By0 = BIT_SET(LocalCAN2Data.T2_By0, 0)
		else
			LocalCAN2Data.T2_By0 = BIT_CLR(LocalCAN2Data.T2_By0, 0)
		endif
	; uiProgrammKategorie
   		LocalCAN2Data.T2_By2_By3	= LocalCOB_Typ_361bis369.uiProgrammKategorie
   	; udKundennummer
	   	 	udShr16 = shr(LocalCOB_Typ_361bis369.udKundennummer,16)
	   	LocalCAN2Data.T2_By4_By5	= UINT(udShr16)									; take UPPERBytes ..
	   	LocalCAN2Data.T2_By6_By7	= UINT(LocalCOB_Typ_361bis369.udKundennummer)	; take LOWER bytes..

	;****ID 361..369****Telegram 3********ID 361..369****Telegram 3********ID 361..369****Telegram 3********ID 361..369****Telegram 3****
		; always set telegram number "01"..
		LocalCAN2Data.T3_By0 = BIT_CLR(LocalCAN2Data.T3_By0, 5)
		LocalCAN2Data.T3_By0 = BIT_SET(LocalCAN2Data.T3_By0, 6)
		; .. and sign CAN2 telegram
		LocalCAN2Data.T3_By0 = BIT_SET(LocalCAN2Data.T3_By0, 7)

      ; ###HO - 270905 - a_usCustomize[0..6]
		if(TARGETInfo_0.DataFormat = 2) then  ; motorola
			memcpy(adr(LocalCAN2Data.T3_By1),adr(LocalCOB_Typ_361bis369.a_usCustomize[0]),1)
			memcpy(adr(LocalCAN2Data.T3_By2_By3),adr(LocalCOB_Typ_361bis369.a_usCustomize[1]),2)
			memcpy(adr(LocalCAN2Data.T3_By4_By5),adr(LocalCOB_Typ_361bis369.a_usCustomize[3]),2)
			memcpy(adr(LocalCAN2Data.T3_By6_By7),adr(LocalCOB_Typ_361bis369.a_usCustomize[5]),2)
		else ; intel
			LocalCAN2Data.T3_By1	 = LocalCOB_Typ_361bis369.a_usCustomize[0]
			LocalCAN2Data.T3_By2_By3 = LocalCOB_Typ_361bis369.a_usCustomize[2] + 256* LocalCOB_Typ_361bis369.a_usCustomize[1]
			LocalCAN2Data.T3_By4_By5 = LocalCOB_Typ_361bis369.a_usCustomize[4] + 256* LocalCOB_Typ_361bis369.a_usCustomize[3]
			LocalCAN2Data.T3_By6_By7 = LocalCOB_Typ_361bis369.a_usCustomize[6] + 256* LocalCOB_Typ_361bis369.a_usCustomize[5]
		endif

	    iStatus = 0
	    pCAN2Data = ADR(LocalCAN2Data)

endaction ; 361..369

;*******action 371bis379********action 371bis379********action 371bis379********action 371bis379********action 371bis379********
action 371..379: ; 371bis379:
    	; pLocalCOB_Typ_371bis379 access Local_InitCAN2PV.pPVData
    	memcpy(adr(LocalCOB_Typ_371bis379),Local_InitCAN2PV.pPVData,sizeof(LocalCOB_Typ_371bis379))

;****ID 371bis379****Telegram 1********ID 371bis379****Telegram 1********ID 371bis379****Telegram 1********ID 371bis379****Telegram 1****
	;T1 mandatotries ->:
		; .. and sign CAN2 telegram
		LocalCAN2Data.T1_By0 = BIT_CLR(LocalCAN2Data.T1_By0, 5)
		LocalCAN2Data.T1_By0 = BIT_CLR(LocalCAN2Data.T1_By0, 6)
		LocalCAN2Data.T1_By0 = BIT_SET(LocalCAN2Data.T1_By0, 7)

	; bDruckstatus
    	if LocalCOB_Typ_371bis379.bDruckstatus = 1 then
			LocalCAN2Data.T1_By0 = BIT_SET(LocalCAN2Data.T1_By0, 0)
		else
			LocalCAN2Data.T1_By0 = BIT_CLR(LocalCAN2Data.T1_By0, 0)
		endif

	; bBereit
    	if LocalCOB_Typ_371bis379.bBereit = 1 then
			LocalCAN2Data.T1_By0 = BIT_SET(LocalCAN2Data.T1_By0, 1)
		else
			LocalCAN2Data.T1_By0 = BIT_CLR(LocalCAN2Data.T1_By0, 1)
		endif

	; usDruckerfehler
		LocalCAN2Data.T1_By1	= LocalCOB_Typ_371bis379.usDruckerfehler
	; usStation
		LocalCAN2Data.T1_By2_By3 = USINT(LocalCOB_Typ_371bis379.usStation) 	; write usStation to lower byte..
		LocalCAN2Data.T1_By2_By3 = shl(LocalCAN2Data.T1_By2_By3,8)			; .. and shift to UPPER byte..

;****ID 371bis379****Telegram 2********ID 371bis379****Telegram 2********ID 371bis379****Telegram 2********ID 371bis379****Telegram 2****
		; always set telegram number "01"..
		LocalCAN2Data.T2_By0 = BIT_SET(LocalCAN2Data.T2_By0, 5)
		LocalCAN2Data.T2_By0 = BIT_CLR(LocalCAN2Data.T2_By0, 6)
		LocalCAN2Data.T2_By0 = BIT_SET(LocalCAN2Data.T2_By0, 7)
		; .. and sign CAN2 telegram

   	; ###HO - 260905 - a_usCustomize[0..6]
		if(TARGETInfo_0.DataFormat = 2) then  ; motorola
			memcpy(adr(LocalCAN2Data.T2_By1),adr(LocalCOB_Typ_371bis379.a_usCustomize[0]),1)
			memcpy(adr(LocalCAN2Data.T2_By2_By3),adr(LocalCOB_Typ_371bis379.a_usCustomize[1]),2)
			memcpy(adr(LocalCAN2Data.T2_By4_By5),adr(LocalCOB_Typ_371bis379.a_usCustomize[3]),2)
			memcpy(adr(LocalCAN2Data.T2_By6_By7),adr(LocalCOB_Typ_371bis379.a_usCustomize[5]),2)
		else ; intel
			LocalCAN2Data.T2_By1	 = LocalCOB_Typ_371bis379.a_usCustomize[0]
			LocalCAN2Data.T2_By2_By3 = LocalCOB_Typ_371bis379.a_usCustomize[2] + 256* LocalCOB_Typ_371bis379.a_usCustomize[1]
			LocalCAN2Data.T2_By4_By5 = LocalCOB_Typ_371bis379.a_usCustomize[4] + 256* LocalCOB_Typ_371bis379.a_usCustomize[3]
			LocalCAN2Data.T2_By6_By7 = LocalCOB_Typ_371bis379.a_usCustomize[6] + 256* LocalCOB_Typ_371bis379.a_usCustomize[5]
		endif

  	iStatus = 0
    pCAN2Data = ADR(LocalCAN2Data)
endaction ; 371bis379

;*******action 401..419********action 401..419********action 401..419********action 401..419********action 401..419********
action 401..419: ; 401..419 :
   	; pLocalCOB_Typ_401bis419 access Local_InitCAN2PV.pPVData
   	memcpy(adr(LocalCOB_Typ_401bis419),Local_InitCAN2PV.pPVData,sizeof(LocalCOB_Typ_401bis419))

;*******action 401..419********action 401..419********action 401..419********action 401..419********action 401..419********

;****ID 401..419****Telegram 1********ID 401..419****Telegram 1********ID 401..419****Telegram 1********ID 401..419****Telegram 1****
;T1 mandatotries ->:
		LocalCAN2Data.T1_By0 = BIT_CLR(LocalCAN2Data.T1_By0, 5)
		LocalCAN2Data.T1_By0 = BIT_CLR(LocalCAN2Data.T1_By0, 6)
		; .. and sign CAN2 telegram
		LocalCAN2Data.T1_By0 = BIT_SET(LocalCAN2Data.T1_By0, 7)

;	++	bBereit
	    if LocalCOB_Typ_401bis419.bBereit = 1 then
			LocalCAN2Data.T1_By0 = BIT_SET(LocalCAN2Data.T1_By0, 0)
		else
			LocalCAN2Data.T1_By0 = BIT_CLR(LocalCAN2Data.T1_By0, 0)
		endif
;	++	bBeladeanforderung
	    if LocalCOB_Typ_401bis419.bBeladeanforderung = 1 then
			LocalCAN2Data.T1_By0 = BIT_SET(LocalCAN2Data.T1_By0, 1)
		else
			LocalCAN2Data.T1_By0 = BIT_CLR(LocalCAN2Data.T1_By0, 1)
		endif
;	++	bEntladefreigabe
	    if LocalCOB_Typ_401bis419.bEntladefreigabe = 1 then
			LocalCAN2Data.T1_By0 = BIT_SET(LocalCAN2Data.T1_By0, 2)
		else
			LocalCAN2Data.T1_By0 = BIT_CLR(LocalCAN2Data.T1_By0, 2)
		endif
;	++	bAnsteuerungSpeicherband
	    if LocalCOB_Typ_401bis419.bAnsteuerungSpeicherband = 1 then
			LocalCAN2Data.T1_By0 = BIT_SET(LocalCAN2Data.T1_By0, 3)
		else
			LocalCAN2Data.T1_By0 = BIT_CLR(LocalCAN2Data.T1_By0, 3)
		endif
		; ###HO 060404 -> ehemals bProgrammabbruch..
;	++	bVorsignal
	    if LocalCOB_Typ_401bis419.bVorsignal = 1 then
			LocalCAN2Data.T1_By0 = BIT_SET(LocalCAN2Data.T1_By0, 4)
		else
			LocalCAN2Data.T1_By0 = BIT_CLR(LocalCAN2Data.T1_By0, 4)
		endif
;	++	udPostennummer
		; broadcast via CAN in 'motorola order' : MSByte as byte2 and LSByte as byte5 !!
			udShr16 = shr(LocalCOB_Typ_401bis419.udPostennummer,16)
    	LocalCAN2Data.T1_By2_By3	= UINT(udShr16)									; take UPPERBytes of Prog/Kat ..
    	LocalCAN2Data.T1_By4_By5	= UINT(LocalCOB_Typ_401bis419.udPostennummer)	; take LOWER byte..
;	++	uiGewicht
	    	LocalCAN2Data.T1_By6_By7	= LocalCOB_Typ_401bis419.uiGewicht

;****ID 401..419****Telegram 2********ID 401..419****Telegram 2********ID 401..419****Telegram 2********ID 401..419****Telegram 2****
;T2 mandatotries ->:
		LocalCAN2Data.T2_By0  					= BIT_SET(LocalCAN2Data.T2_By0, 5)
		LocalCAN2Data.T2_By0  					= BIT_CLR(LocalCAN2Data.T2_By0, 6)
		; .. and sign CAN2 telegram
		LocalCAN2Data.T2_By0 					= BIT_SET(LocalCAN2Data.T2_By0, 7)
;  	++	bProgrammOderKategorie
	    if LocalCOB_Typ_401bis419.bProgrammOderKategorie = 1 then
			LocalCAN2Data.T2_By0 = BIT_SET(LocalCAN2Data.T2_By0, 0)
		else
			LocalCAN2Data.T2_By0 = BIT_CLR(LocalCAN2Data.T2_By0, 0)
		endif
	; ###HO - 310805 -  bFreigabeFlusen
		if LocalCOB_Typ_401bis419.bFreigabeFlusen = 1 then
			LocalCAN2Data.T2_By0 = BIT_SET(LocalCAN2Data.T2_By0, 1)
		else
			LocalCAN2Data.T2_By0 = BIT_CLR(LocalCAN2Data.T2_By0, 1)
		endif
;	++	bKippsperre
	    if LocalCOB_Typ_401bis419.bKippsperre = 1 then
			LocalCAN2Data.T2_By0 = BIT_SET(LocalCAN2Data.T2_By0, 2)
		else
			LocalCAN2Data.T2_By0 = BIT_CLR(LocalCAN2Data.T2_By0, 2)
		endif
   ; bNotAusVerbST
	    if LocalCOB_Typ_401bis419.bNotAusVerbST = 1 then
			LocalCAN2Data.T2_By0 = BIT_SET(LocalCAN2Data.T2_By0, 4)
		else
			LocalCAN2Data.T2_By0 = BIT_CLR(LocalCAN2Data.T2_By0, 4)
		endif
;	++	uiProgrammKategorie
	    	LocalCAN2Data.T2_By2_By3	= LocalCOB_Typ_401bis419.uiProgrammKategorie
;	++	udKundennummer
			udShr16 = shr(LocalCOB_Typ_401bis419.udKundennummer,16)
    	LocalCAN2Data.T2_By4_By5	= UINT(udShr16)									; take UPPERBytes of Prog/Kat ..
    	LocalCAN2Data.T2_By6_By7	= UINT(LocalCOB_Typ_401bis419.udKundennummer)	; take LOWER byte..

;****ID 401..419****Telegram 3********ID 401..419****Telegram 3********ID 401..419****Telegram 3*****
;T3 mandatotries ->:
	LocalCAN2Data.T3_By0 = BIT_CLR(LocalCAN2Data.T3_By0, 5)
	LocalCAN2Data.T3_By0 = BIT_SET(LocalCAN2Data.T3_By0, 6)
	; .. and sign CAN2 telegram
	LocalCAN2Data.T3_By0 = BIT_SET(LocalCAN2Data.T3_By0, 7)

      ; ###HO - 270905 - a_usCustomize[0..6]
		if(TARGETInfo_0.DataFormat = 2) then  ; motorola
			memcpy(adr(LocalCAN2Data.T3_By1),adr(LocalCOB_Typ_401bis419.a_usCustomize[0]),1)
			memcpy(adr(LocalCAN2Data.T3_By2_By3),adr(LocalCOB_Typ_401bis419.a_usCustomize[1]),2)
			memcpy(adr(LocalCAN2Data.T3_By4_By5),adr(LocalCOB_Typ_401bis419.a_usCustomize[3]),2)
			memcpy(adr(LocalCAN2Data.T3_By6_By7),adr(LocalCOB_Typ_401bis419.a_usCustomize[5]),2)
		else ; intel
			LocalCAN2Data.T3_By1	 = LocalCOB_Typ_401bis419.a_usCustomize[0]
			LocalCAN2Data.T3_By2_By3 = LocalCOB_Typ_401bis419.a_usCustomize[2] + 256* LocalCOB_Typ_401bis419.a_usCustomize[1]
			LocalCAN2Data.T3_By4_By5 = LocalCOB_Typ_401bis419.a_usCustomize[4] + 256* LocalCOB_Typ_401bis419.a_usCustomize[3]
			LocalCAN2Data.T3_By6_By7 = LocalCOB_Typ_401bis419.a_usCustomize[6] + 256* LocalCOB_Typ_401bis419.a_usCustomize[5]
		endif

    iStatus = 0
    pCAN2Data = ADR(LocalCAN2Data)
endaction ; 401..419

;*******action 421********action 421********action 421********action 421********action 421********
action 421..439: ; 421:
   	; pLocalCOB_Typ_421bis439 access Local_InitCAN2PV.pPVData
   	memcpy(adr(LocalCOB_Typ_421bis439),Local_InitCAN2PV.pPVData,sizeof(LocalCOB_Typ_421bis439))

;****ID 421****Telegram 1********ID 421****Telegram 1********ID 421****Telegram 1********ID 421****Telegram 1****
;T1 mandatotries ->:
		LocalCAN2Data.T1_By1 = BIT_CLR(LocalCAN2Data.T1_By1, 3)
		LocalCAN2Data.T1_By1 = BIT_CLR(LocalCAN2Data.T1_By1, 4)
		; .. and sign CAN2 telegram
		LocalCAN2Data.T1_By1 = BIT_SET(LocalCAN2Data.T1_By1, 5)

	; bBereit					1
		if LocalCOB_Typ_421bis439.bBereit = 1 then
			LocalCAN2Data.T1_By0 = BIT_SET(LocalCAN2Data.T1_By0, 0)
		else
			LocalCAN2Data.T1_By0 = BIT_CLR(LocalCAN2Data.T1_By0, 0)
		endif
	; bBeladebereit					1
		if LocalCOB_Typ_421bis439.bBeladebereit = 1 then
			LocalCAN2Data.T1_By0 = BIT_SET(LocalCAN2Data.T1_By0, 1)
		else
			LocalCAN2Data.T1_By0 = BIT_CLR(LocalCAN2Data.T1_By0, 1)
		endif
	; bBelaedt						1
		if LocalCOB_Typ_421bis439.bBelaedt = 1 then
			LocalCAN2Data.T1_By0 = BIT_SET(LocalCAN2Data.T1_By0, 2)
		else
			LocalCAN2Data.T1_By0 = BIT_CLR(LocalCAN2Data.T1_By0, 2)
		endif
	; bEntladebereit					1
		if LocalCOB_Typ_421bis439.bEntladebereit = 1 then
			LocalCAN2Data.T1_By0 = BIT_SET(LocalCAN2Data.T1_By0, 3)
		else
			LocalCAN2Data.T1_By0 = BIT_CLR(LocalCAN2Data.T1_By0, 3)
		endif
	; ###060404 umbenannt von 'bEntlaedt'
	; bEntlade						1
		if LocalCOB_Typ_421bis439.bEntlade = 1 then
			LocalCAN2Data.T1_By0 = BIT_SET(LocalCAN2Data.T1_By0, 4)
		else
			LocalCAN2Data.T1_By0 = BIT_CLR(LocalCAN2Data.T1_By0, 4)
		endif
	; bTrocknet						1
		if LocalCOB_Typ_421bis439.bTrocknet = 1 then
			LocalCAN2Data.T1_By1 = BIT_SET(LocalCAN2Data.T1_By1, 1)
		else
			LocalCAN2Data.T1_By1 = BIT_CLR(LocalCAN2Data.T1_By1, 1)
		endif
	; bHauptgeblaese					1
		if LocalCOB_Typ_421bis439.bHauptgeblaese = 1 then
			LocalCAN2Data.T1_By0 = BIT_SET(LocalCAN2Data.T1_By0, 6)
		else
			LocalCAN2Data.T1_By0 = BIT_CLR(LocalCAN2Data.T1_By0, 6)
		endif
	; bFlusenabsaugung				1
		if LocalCOB_Typ_421bis439.bFlusenabsaugung = 1 then
			LocalCAN2Data.T1_By0 = BIT_SET(LocalCAN2Data.T1_By0, 7)
		else
			LocalCAN2Data.T1_By0 = BIT_CLR(LocalCAN2Data.T1_By0, 7)
		endif
	; bAbkuehlung						1
		if LocalCOB_Typ_421bis439.bAbkuehlung = 1 then
			LocalCAN2Data.T1_By1 = BIT_SET(LocalCAN2Data.T1_By1, 2)
		else
			LocalCAN2Data.T1_By1 = BIT_CLR(LocalCAN2Data.T1_By1, 2)
		endif
	; bLichtschrSpeicherbandHinten	1
		if LocalCOB_Typ_421bis439.bLichtschrSpeicherbandHinten = 1 then
			LocalCAN2Data.T1_By1 = BIT_SET(LocalCAN2Data.T1_By1, 6)
		else
			LocalCAN2Data.T1_By1 = BIT_CLR(LocalCAN2Data.T1_By1, 6)
		endif
	; bLichtschrSpeicherbandVorne		1
		if LocalCOB_Typ_421bis439.bLichtschrSpeicherbandVorne = 1 then
			LocalCAN2Data.T1_By1 = BIT_SET(LocalCAN2Data.T1_By1, 7)
		else
			LocalCAN2Data.T1_By1 = BIT_CLR(LocalCAN2Data.T1_By1, 7)
		endif
	; bEIN							1
		if LocalCOB_Typ_421bis439.bEIN = 1 then
			LocalCAN2Data.T1_By1 = BIT_SET(LocalCAN2Data.T1_By1, 0)
		else
			LocalCAN2Data.T1_By1 = BIT_CLR(LocalCAN2Data.T1_By1, 0)
		endif
	; bStoerung						1
		if LocalCOB_Typ_421bis439.bStoerung = 1 then
			LocalCAN2Data.T1_By0 = BIT_SET(LocalCAN2Data.T1_By0, 5)
		else
			LocalCAN2Data.T1_By0 = BIT_CLR(LocalCAN2Data.T1_By0, 5)
		endif
	; udPostennummer					1
		; broadcast via CAN in 'motorola order' : MSByte as byte2 and LSByte as byte5 !!
			udShr16 = shr(LocalCOB_Typ_421bis439.udPostennummer,16)
    	LocalCAN2Data.T1_By2_By3	= UINT(udShr16)									; take UPPERBytes of Prog/Kat ..
    	LocalCAN2Data.T1_By4_By5	= UINT(LocalCOB_Typ_421bis439.udPostennummer)	; take LOWER byte..
	; uiGewicht						1
		LocalCAN2Data.T1_By6_By7 = LocalCOB_Typ_421bis439.uiGewicht

;****ID 421****Telegram 2********ID 421****Telegram 2********ID 421****Telegram 2********ID 421****Telegram 2****
;T2 mandatotries ->:
		LocalCAN2Data.T2_By1			= BIT_SET(LocalCAN2Data.T2_By1, 3)
		LocalCAN2Data.T2_By1  			= BIT_CLR(LocalCAN2Data.T2_By1, 4)
		; .. and sign CAN2 telegram
		LocalCAN2Data.T2_By1 			= BIT_SET(LocalCAN2Data.T2_By1, 5)
	; bProgrammOderKategorie
		if LocalCOB_Typ_421bis439.bProgrammOderKategorie = 1 then
			LocalCAN2Data.T2_By1 = BIT_SET(LocalCAN2Data.T2_By1, 0)
		else
			LocalCAN2Data.T2_By1 = BIT_CLR(LocalCAN2Data.T2_By1, 0)
		endif
	; bHand
		if LocalCOB_Typ_421bis439.bHand = 1 then
			LocalCAN2Data.T2_By0 = BIT_SET(LocalCAN2Data.T2_By0, 0)
		else
			LocalCAN2Data.T2_By0 = BIT_CLR(LocalCAN2Data.T2_By0, 0)
		endif
		; ###HO 060404 bNotAus umbenannt in bNotAusTrockner
	; bNotAusTrockner
		if LocalCOB_Typ_421bis439.bNotAusTrockner = 1 then
			LocalCAN2Data.T2_By0 = BIT_SET(LocalCAN2Data.T2_By0, 6)
		else
			LocalCAN2Data.T2_By0 = BIT_CLR(LocalCAN2Data.T2_By0, 6)
		endif
	; uiProgrammKategorie
		LocalCAN2Data.T2_By2_By3 = LocalCOB_Typ_421bis439.uiProgrammKategorie
	; udKundennummer
		; broadcast via CAN in 'motorola order' : MSByte as byte2 and LSByte as byte5 !!
			udShr16 = shr(LocalCOB_Typ_421bis439.udKundennummer,16)
    	LocalCAN2Data.T2_By4_By5	= UINT(udShr16)								; take UPPERBytes of Prog/Kat ..
    	LocalCAN2Data.T2_By6_By7	= UINT(LocalCOB_Typ_421bis439.udKundennummer)	; take LOWER byte..

;****ID 421****Telegram 3********ID 421****Telegram 3********ID 421****Telegram 3********ID 421****Telegram 3****
;T3 mandatotries ->:
		LocalCAN2Data.T3_By1  			= BIT_CLR(LocalCAN2Data.T3_By1, 3)
		LocalCAN2Data.T3_By1			= BIT_SET(LocalCAN2Data.T3_By1, 4)
		; .. and sign CAN2 telegram
		LocalCAN2Data.T3_By1 			= BIT_SET(LocalCAN2Data.T3_By1, 5)

	; bTemperatureinheit
		if LocalCOB_Typ_421bis439.bTemperatureinheit = 1 then
			LocalCAN2Data.T3_By1 = BIT_SET(LocalCAN2Data.T3_By1, 7)
		else
			LocalCAN2Data.T3_By1 = BIT_CLR(LocalCAN2Data.T3_By1, 7)
		endif
	; uiRestzeit
		LocalCAN2Data.T3_By2_By3	= LocalCOB_Typ_421bis439.uiRestzeit

	; ###HO 060404  usZulufttemperatur + usAbluftIRTemp entfallen
	;				- dafür uiAbluftTemp + uiIRTemp
(*
	; usZulufttemperatur -> By4 +  usAbluftIRTemp ->  By5
		; set two single bytes to WORD .. -> this matches!!
		; set CAN byte 4..
		LocalCAN2Data.T3_By4_By5	= UINT(LocalCOB_Typ_421bis439.usZulufttemperatur)	; set to LOWER byte..
			uiShl8 = shl(LocalCAN2Data.T3_By4_By5,8)									; .. and shift to UPPER byte..
		; set CAN byte 5..
		LocalCAN2Data.T3_By4_By5 = uiShl8 + LocalCOB_Typ_421bis439.usAbluftIRTemp		; add LOWER byte..
*)
		LocalCAN2Data.T3_By4_By5 = LocalCOB_Typ_421bis439.uiAbluftTemp
		LocalCAN2Data.T3_By6_By7 = LocalCOB_Typ_421bis439.uiIRTemp

;****ID 421****Telegram 4********ID 421****Telegram 4********ID 421****Telegram 4********ID 421****Telegram 4****
;T4 mandatotries ->:
		LocalCAN2Data.T4_By1			= BIT_SET(LocalCAN2Data.T4_By1, 3)
		LocalCAN2Data.T4_By1  			= BIT_SET(LocalCAN2Data.T4_By1, 4)
		; .. and sign CAN2 telegram
		LocalCAN2Data.T4_By1 			= BIT_SET(LocalCAN2Data.T4_By1, 5)

  	; ###HO - 260905 - a_usCustomize[0..6]
		if(TARGETInfo_0.DataFormat = 2) then  ; motorola
			memcpy(adr(LocalCAN2Data.T4_By0),adr(LocalCOB_Typ_421bis439.a_usCustomize[0]),1)
			memcpy(adr(LocalCAN2Data.T4_By2_By3),adr(LocalCOB_Typ_421bis439.a_usCustomize[1]),2)
			memcpy(adr(LocalCAN2Data.T4_By4_By5),adr(LocalCOB_Typ_421bis439.a_usCustomize[3]),2)
			memcpy(adr(LocalCAN2Data.T4_By6_By7),adr(LocalCOB_Typ_421bis439.a_usCustomize[5]),2)
		else ; intel
			LocalCAN2Data.T4_By0	 = LocalCOB_Typ_421bis439.a_usCustomize[0]
			LocalCAN2Data.T4_By2_By3 = LocalCOB_Typ_421bis439.a_usCustomize[2] + 256* LocalCOB_Typ_421bis439.a_usCustomize[1]
			LocalCAN2Data.T4_By4_By5 = LocalCOB_Typ_421bis439.a_usCustomize[4] + 256* LocalCOB_Typ_421bis439.a_usCustomize[3]
			LocalCAN2Data.T4_By6_By7 = LocalCOB_Typ_421bis439.a_usCustomize[6] + 256* LocalCOB_Typ_421bis439.a_usCustomize[5]
		endif

	; Telegrammabschluss markieren..
    iStatus = 0
    pCAN2Data = ADR(LocalCAN2Data)
endaction ; 421

;*******action 441..459********action 441..459********action 441..459********action 441..459********action 441..459********
action 441..459: ; 441..459:
    	; pLocalCOB_Typ_441bis459 access Local_InitCAN2PV.pPVData
    	memcpy(adr(LocalCOB_Typ_441bis459),Local_InitCAN2PV.pPVData,sizeof(LocalCOB_Typ_441bis459))

;****ID 441..459****Telegram 1********ID 441..459****Telegram 1********ID 441..459****Telegram 1********ID 441..459****Telegram 1****
	;T1 mandatotries ->:
	;	..über temp-Byte gehen - By2_3 teilen sich Nutzdaten + Mandatories..
	; 	Byte3 z.Zt. leer..
		usTempBy2 = 0
		usTempBy2 = BIT_CLR(usTempBy2,6)
		usTempBy2 = BIT_SET(usTempBy2,7); .. and sign CAN2 telegram

	; ###HO - 310805 - bVorsignal Flusen
		if LocalCOB_Typ_441bis459.bVorsignalFlusen = 1 then
			usTempBy2 = BIT_SET(usTempBy2, 0)
		else
			usTempBy2 = BIT_CLR(usTempBy2, 0)
		endif
	; ###HO - 310805 - bSaugbeladungAktiv
		if LocalCOB_Typ_441bis459.bSaugbeladungAktiv = 1 then
			usTempBy2 = BIT_SET(usTempBy2, 1)
		else
			usTempBy2 = BIT_CLR(usTempBy2, 1)
		endif
	; ###HO - 310805 - bAnforderungFlusen
		if LocalCOB_Typ_441bis459.bAnforderungFlusen = 1 then
			usTempBy2 = BIT_SET(usTempBy2, 2)
		else
			usTempBy2 = BIT_CLR(usTempBy2, 2)
		endif

	; Byte2 an die richtige Stelle schieben..
	LocalCAN2Data.T1_By2_By3 = UINT(usTempBy2)
	if(TARGETInfo_0.DataFormat = 2) then  ; m68k
		LocalCAN2Data.T1_By2_By3 = shl(LocalCAN2Data.T1_By2_By3,8)
	else ; i386
		; nicht shiften..
		LocalCAN2Data.T1_By2_By3 = shl(LocalCAN2Data.T1_By2_By3,8)
	endif

	; uiTrocknerrestzeit
   		if(TARGETInfo_0.DataFormat = 2) then  ; m68k
			LocalCAN2Data.T1_By0 = USINT(shr(LocalCOB_Typ_441bis459.uiTrocknerrestzeit,8))
			LocalCAN2Data.T1_By1 = USINT(LocalCOB_Typ_441bis459.uiTrocknerrestzeit)
		else ; i386
			LocalCAN2Data.T1_By0 = USINT(shr(LocalCOB_Typ_441bis459.uiTrocknerrestzeit,8))
			LocalCAN2Data.T1_By1 = USINT(LocalCOB_Typ_441bis459.uiTrocknerrestzeit)
		endif

;****ID 441..459****Telegram 2********ID 441..459****Telegram 2********ID 441..459****Telegram 2********ID 441..459****Telegram 2****
	;T2 mandatotries ->:
	; LocalCAN2Data.T2_By2_By3 -> dieses WORT teilen sich Steuerbyte+Nutzinfos..
	usTempBy2 = 0
	usTempBy2 = BIT_SET(usTempBy2,6)
	usTempBy2 = BIT_SET(usTempBy2,7); .. and sign CAN2 telegram

	usTempBy3 = LocalCOB_Typ_441bis459.a_usCustomize[2]

	; Bytes 2+3 an die richtige Stelle schieben..
	LocalCAN2Data.T2_By2_By3 = UINT(usTempBy2)
	if(TARGETInfo_0.DataFormat = 2) then  ; m68k
		LocalCAN2Data.T2_By2_By3 = shl(LocalCAN2Data.T2_By2_By3,8)
		LocalCAN2Data.T2_By2_By3= LocalCAN2Data.T2_By2_By3 + usTempBy3
	else ; i386
		LocalCAN2Data.T2_By2_By3 = shl(LocalCAN2Data.T2_By2_By3,8)
		LocalCAN2Data.T2_By2_By3= LocalCAN2Data.T2_By2_By3 + usTempBy3
	endif

		; das Steuerbyte liegt inmitten der Daten..
		; Targetunabhängig - nur USINTs
		memcpy(adr(LocalCAN2Data.T2_By0), adr(LocalCOB_Typ_441bis459.a_usCustomize[0]),2)

	; ###HO - 260905 - a_usCustomize[0..6]
		if(TARGETInfo_0.DataFormat = 2) then  ; motorola
			; LocalCAN2Data.T2_By2_By3 -> s.o.
			memcpy(adr(LocalCAN2Data.T2_By4_By5), adr(LocalCOB_Typ_441bis459.a_usCustomize[3]),2)
			memcpy(adr(LocalCAN2Data.T2_By6_By7), adr(LocalCOB_Typ_441bis459.a_usCustomize[5]),2)
		else ; intel
			LocalCAN2Data.T2_By4_By5 = LocalCOB_Typ_441bis459.a_usCustomize[4] + 256* LocalCOB_Typ_441bis459.a_usCustomize[3]
			LocalCAN2Data.T2_By6_By7 = LocalCOB_Typ_441bis459.a_usCustomize[6] + 256* LocalCOB_Typ_441bis459.a_usCustomize[5]
		endif

    iStatus = 0
    pCAN2Data = ADR(LocalCAN2Data)
endaction ; 441..459

;*******action 480********action 480********action 480********action 480********action 480********
action 480:
	    ; to do: transform LocalHFAnWaschm_ObjNr120_type data to LocalCAN2Data
  		memcpy(adr(LocalCOB_Typ_480),Local_InitCAN2PV.pPVData,sizeof(LocalCOB_Typ_480))

;****ID 480****Telegram 1********ID 480****Telegram 1********ID 480****Telegram 1********ID 480****Telegram 1****
;T1 mandatotries ->:
		LocalCAN2Data.T1_By0 = BIT_CLR(LocalCAN2Data.T1_By0, 5)
		LocalCAN2Data.T1_By0 = BIT_CLR(LocalCAN2Data.T1_By0, 6)
		; .. and sign CAN2 telegram
		LocalCAN2Data.T1_By0 = BIT_SET(LocalCAN2Data.T1_By0, 7)
;----------------------------By 0--------------------------------------
; bBereit
		if LocalCOB_Typ_480.bBereit = 1 then
			LocalCAN2Data.T1_By0 = BIT_SET(LocalCAN2Data.T1_By0, 0)
		else
			LocalCAN2Data.T1_By0 = BIT_CLR(LocalCAN2Data.T1_By0, 0)
		endif
; bBeladebereit
		if LocalCOB_Typ_480.bBeladebereit = 1 then
			LocalCAN2Data.T1_By0 = BIT_SET(LocalCAN2Data.T1_By0, 1)
		else
			LocalCAN2Data.T1_By0 = BIT_CLR(LocalCAN2Data.T1_By0, 1)
		endif
; bBeladungAktiv
		if LocalCOB_Typ_480.bBeladungAktiv = 1 then
			LocalCAN2Data.T1_By0 = BIT_SET(LocalCAN2Data.T1_By0, 2)
		else
			LocalCAN2Data.T1_By0 = BIT_CLR(LocalCAN2Data.T1_By0, 2)
		endif
; bStörung
		if LocalCOB_Typ_480.bStoerung = 1 then
			LocalCAN2Data.T1_By0 = BIT_SET(LocalCAN2Data.T1_By0, 3)
		else
			LocalCAN2Data.T1_By0 = BIT_CLR(LocalCAN2Data.T1_By0, 3)
		endif
; bBeladeanfHalbauto
		if LocalCOB_Typ_480.bBeladeanfHalbauto = 1 then
			LocalCAN2Data.T1_By0 = BIT_SET(LocalCAN2Data.T1_By0, 4)
		else
			LocalCAN2Data.T1_By0 = BIT_CLR(LocalCAN2Data.T1_By0, 4)
		endif
;----------------------------By 1--------------------------------------
; bBeladeabbruch
		if LocalCOB_Typ_480.bBeladeabbruch = 1 then
			LocalCAN2Data.T1_By1 = BIT_SET(LocalCAN2Data.T1_By1, 0)
		else
			LocalCAN2Data.T1_By1 = BIT_CLR(LocalCAN2Data.T1_By1, 0)
		endif
; bFreigabeBeladung
		if LocalCOB_Typ_480.bFreigabeBeladung = 1 then
			LocalCAN2Data.T1_By1 = BIT_SET(LocalCAN2Data.T1_By1, 1)
		else
			LocalCAN2Data.T1_By1 = BIT_CLR(LocalCAN2Data.T1_By1, 1)
		endif
; bDurchschleusenStart
		if LocalCOB_Typ_480.bDurchschleusenStart = 1 then
			LocalCAN2Data.T1_By1 = BIT_SET(LocalCAN2Data.T1_By1, 2)
		else
			LocalCAN2Data.T1_By1 = BIT_CLR(LocalCAN2Data.T1_By1, 2)
		endif
; bNotAusAero
		if LocalCOB_Typ_480.bNotAusAero = 1 then
			LocalCAN2Data.T1_By1 = BIT_SET(LocalCAN2Data.T1_By1, 3)
		else
			LocalCAN2Data.T1_By1 = BIT_CLR(LocalCAN2Data.T1_By1, 3)
		endif
; bBeladepause
		if LocalCOB_Typ_480.bBeladepause = 1 then
			LocalCAN2Data.T1_By1 = BIT_SET(LocalCAN2Data.T1_By1, 4)
		else
			LocalCAN2Data.T1_By1 = BIT_CLR(LocalCAN2Data.T1_By1, 4)
		endif
; T1-By - 5..7 -> Redundanzen..
		if LocalCOB_Typ_480.bReserve1 = 1 then
			LocalCAN2Data.T1_By1 = BIT_SET(LocalCAN2Data.T1_By1, 5)
		else
			LocalCAN2Data.T1_By1 = BIT_CLR(LocalCAN2Data.T1_By1, 5)
		endif
		if LocalCOB_Typ_480.bReserve2 = 1 then
			LocalCAN2Data.T1_By1 = BIT_SET(LocalCAN2Data.T1_By1, 6)
		else
			LocalCAN2Data.T1_By1 = BIT_CLR(LocalCAN2Data.T1_By1, 6)
		endif
		if LocalCOB_Typ_480.bReserve3 = 1 then
			LocalCAN2Data.T1_By1 = BIT_SET(LocalCAN2Data.T1_By1, 7)
		else
			LocalCAN2Data.T1_By1 = BIT_CLR(LocalCAN2Data.T1_By1, 7)
		endif
; udPostennummer						1
			udShr16 = shr(LocalCOB_Typ_480.udPostennummer,16)
    	LocalCAN2Data.T1_By2_By3	= UINT(udShr16)							; take UPPERBytes of Prog/Kat ..
    	LocalCAN2Data.T1_By4_By5	= UINT(LocalCOB_Typ_480.udPostennummer)	; take LOWER byte..
; uiGewicht						1
		LocalCAN2Data.T1_By6_By7 = LocalCOB_Typ_480.uiGewicht

;****ID 480****Telegram 2********ID 480****Telegram 2********ID 480****Telegram 2********ID 480****Telegram 2****
;T2 mandatotries ->:
		LocalCAN2Data.T2_By0 		= BIT_SET(LocalCAN2Data.T2_By0, 5)
		LocalCAN2Data.T2_By0 		= BIT_CLR(LocalCAN2Data.T2_By0, 6)
		; .. and sign CAN2 telegram
		LocalCAN2Data.T2_By0 		= BIT_SET(LocalCAN2Data.T2_By0, 7)

; bProgKat
		if LocalCOB_Typ_480.bProgKat = 1 then
			LocalCAN2Data.T2_By0 = BIT_SET(LocalCAN2Data.T2_By0, 0)
		else
			LocalCAN2Data.T2_By0 = BIT_CLR(LocalCAN2Data.T2_By0, 0)
		endif
; Redundanzen -> T2-By0 - bit1..5
		if LocalCOB_Typ_480.bReserve4 = 1 then
			LocalCAN2Data.T2_By0 = BIT_SET(LocalCAN2Data.T2_By0, 1)
		else
			LocalCAN2Data.T2_By0 = BIT_CLR(LocalCAN2Data.T2_By0, 1)
		endif
		if LocalCOB_Typ_480.bReserve5 = 1 then
			LocalCAN2Data.T2_By0 = BIT_SET(LocalCAN2Data.T2_By0, 2)
		else
			LocalCAN2Data.T2_By0 = BIT_CLR(LocalCAN2Data.T2_By0, 2)
		endif
		if LocalCOB_Typ_480.bReserve6 = 1 then
			LocalCAN2Data.T2_By0 = BIT_SET(LocalCAN2Data.T2_By0, 3)
		else
			LocalCAN2Data.T2_By0 = BIT_CLR(LocalCAN2Data.T2_By0, 3)
		endif
		if LocalCOB_Typ_480.bReserve7 = 1 then
			LocalCAN2Data.T2_By0 = BIT_SET(LocalCAN2Data.T2_By0, 4)
		else
			LocalCAN2Data.T2_By0 = BIT_CLR(LocalCAN2Data.T2_By0, 4)
		endif
;Redundanzen
		LocalCAN2Data.T2_By1 = LocalCOB_Typ_480.usReserve1
; uiProgKat
		LocalCAN2Data.T2_By2_By3 = LocalCOB_Typ_480.uiProgKat
; udKundennummer
			udShr16 = shr(LocalCOB_Typ_480.udKundennummer,16)
    	LocalCAN2Data.T2_By4_By5	= UINT(udShr16)							; take UPPERBytes of Prog/Kat ..
    	LocalCAN2Data.T2_By6_By7	= UINT(LocalCOB_Typ_480.udKundennummer)	; take LOWER byte..

;****ID 480****Telegram 3********ID 480****Telegram 3********ID 480****Telegram 3********ID 480****Telegram 3****
;T3 mandatotries ->:
	LocalCAN2Data.T3_By0 		= BIT_CLR(LocalCAN2Data.T3_By0, 5)
	LocalCAN2Data.T3_By0 		= BIT_SET(LocalCAN2Data.T3_By0, 6)
	; .. and sign CAN2 telegram
	LocalCAN2Data.T3_By0 		= BIT_SET(LocalCAN2Data.T3_By0, 7)

; 	Res 8..9
		if LocalCOB_Typ_480.bReserve8 = 1 then
			LocalCAN2Data.T3_By0 = BIT_SET(LocalCAN2Data.T3_By0, 0)
		else
			LocalCAN2Data.T3_By0 = BIT_CLR(LocalCAN2Data.T3_By0, 0)
		endif
		if LocalCOB_Typ_480.bReserve9 = 1 then
			LocalCAN2Data.T3_By0 = BIT_SET(LocalCAN2Data.T3_By0, 1)
		else
			LocalCAN2Data.T3_By0 = BIT_CLR(LocalCAN2Data.T3_By0, 1)
		endif

	; ###HO - 260905 - a_usCustomize[0..6]
		if(TARGETInfo_0.DataFormat = 2) then  ; motorola
			memcpy(adr(LocalCAN2Data.T3_By1),adr(LocalCOB_Typ_480.a_usCustomize[0]),1)
			memcpy(adr(LocalCAN2Data.T3_By2_By3),adr(LocalCOB_Typ_480.a_usCustomize[1]),2)
			memcpy(adr(LocalCAN2Data.T3_By4_By5),adr(LocalCOB_Typ_480.a_usCustomize[3]),2)
			memcpy(adr(LocalCAN2Data.T3_By6_By7),adr(LocalCOB_Typ_480.a_usCustomize[5]),2)
		else ; intel
			LocalCAN2Data.T3_By1	 = LocalCOB_Typ_480.a_usCustomize[0]
			LocalCAN2Data.T3_By2_By3 = LocalCOB_Typ_480.a_usCustomize[2] + 256* LocalCOB_Typ_480.a_usCustomize[1]
			LocalCAN2Data.T3_By4_By5 = LocalCOB_Typ_480.a_usCustomize[4] + 256* LocalCOB_Typ_480.a_usCustomize[3]
			LocalCAN2Data.T3_By6_By7 = LocalCOB_Typ_480.a_usCustomize[6] + 256* LocalCOB_Typ_480.a_usCustomize[5]
		endif

	iStatus = 0
	pCAN2Data = ADR(LocalCAN2Data)
endaction ; ID 480

;*******action 481********action 481********action 481********action 481********action 481********
action 481:
	    ; to do: transform LocalHFAnWaschm_ObjNr120_type data to LocalCAN2Data
  		memcpy(adr(LocalCOB_Typ_481),Local_InitCAN2PV.pPVData,sizeof(LocalCOB_Typ_481))

;****ID 481****Telegram 1********ID 481****Telegram 1********ID 481****Telegram 1********ID 481****Telegram 1****
;T1 mandatotries ->:
	LocalCAN2Data.T1_By0 = BIT_CLR(LocalCAN2Data.T1_By0, 5)
	LocalCAN2Data.T1_By0 = BIT_CLR(LocalCAN2Data.T1_By0, 6)
	; .. and sign CAN2 telegram
	LocalCAN2Data.T1_By0 = BIT_SET(LocalCAN2Data.T1_By0, 7)

; bBereit
		if LocalCOB_Typ_481.bBereit = 1 then
			LocalCAN2Data.T1_By0 = BIT_SET(LocalCAN2Data.T1_By0, 0)
		else
			LocalCAN2Data.T1_By0 = BIT_CLR(LocalCAN2Data.T1_By0, 0)
		endif
; bBeladeanfAuto
		if LocalCOB_Typ_481.bBeladeanfAuto = 1 then
			LocalCAN2Data.T1_By0 = BIT_SET(LocalCAN2Data.T1_By0, 1)
		else
			LocalCAN2Data.T1_By0 = BIT_CLR(LocalCAN2Data.T1_By0, 1)
		endif
; bStoerung
		if LocalCOB_Typ_481.bStoerung = 1 then
			LocalCAN2Data.T1_By0 = BIT_SET(LocalCAN2Data.T1_By0, 2)
		else
			LocalCAN2Data.T1_By0 = BIT_CLR(LocalCAN2Data.T1_By0, 2)
		endif
; bAnlagenstrgHalbauto
		if LocalCOB_Typ_481.bAnlagenstrgHalbauto = 1 then
			LocalCAN2Data.T1_By0 = BIT_SET(LocalCAN2Data.T1_By0, 3)
		else
			LocalCAN2Data.T1_By0 = BIT_CLR(LocalCAN2Data.T1_By0, 3)
		endif
; bAnlagenstrgAuto
		if LocalCOB_Typ_481.bAnlagenstrgAuto = 1 then
			LocalCAN2Data.T1_By0 = BIT_SET(LocalCAN2Data.T1_By0, 4)
		else
			LocalCAN2Data.T1_By0 = BIT_CLR(LocalCAN2Data.T1_By0, 4)
		endif
; bDurchschleusen
		if LocalCOB_Typ_481.bDurchschleusen = 1 then
			LocalCAN2Data.T1_By1 = BIT_SET(LocalCAN2Data.T1_By1, 0)
		else
			LocalCAN2Data.T1_By1 = BIT_CLR(LocalCAN2Data.T1_By1, 0)
		endif
; bFreigabeDurchschl
		if LocalCOB_Typ_481.bFreigabeDurchschl = 1 then
			LocalCAN2Data.T1_By1 = BIT_SET(LocalCAN2Data.T1_By1, 1)
		else
			LocalCAN2Data.T1_By1 = BIT_CLR(LocalCAN2Data.T1_By1, 1)
		endif
; bNotAusAnlagenStrg
		if LocalCOB_Typ_481.bNotAusAnlagenStrg = 1 then
			LocalCAN2Data.T1_By1 = BIT_SET(LocalCAN2Data.T1_By1, 2)
		else
			LocalCAN2Data.T1_By1 = BIT_CLR(LocalCAN2Data.T1_By1, 2)
		endif
; bPauseAktiv
		if LocalCOB_Typ_481.bPauseAktiv = 1 then
			LocalCAN2Data.T1_By1 = BIT_SET(LocalCAN2Data.T1_By1, 3)
		else
			LocalCAN2Data.T1_By1 = BIT_CLR(LocalCAN2Data.T1_By1, 3)
		endif
; T1-By - 3..7 -> Redundanzen..
		if LocalCOB_Typ_481.bReserve1 = 1 then
			LocalCAN2Data.T1_By1 = BIT_SET(LocalCAN2Data.T1_By1, 4)
		else
			LocalCAN2Data.T1_By1 = BIT_CLR(LocalCAN2Data.T1_By1, 4)
		endif
		if LocalCOB_Typ_481.bReserve2 = 1 then
			LocalCAN2Data.T1_By1 = BIT_SET(LocalCAN2Data.T1_By1, 5)
		else
			LocalCAN2Data.T1_By1 = BIT_CLR(LocalCAN2Data.T1_By1, 5)
		endif
		if LocalCOB_Typ_481.bReserve3 = 1 then
			LocalCAN2Data.T1_By1 = BIT_SET(LocalCAN2Data.T1_By1, 6)
		else
			LocalCAN2Data.T1_By1 = BIT_CLR(LocalCAN2Data.T1_By1, 6)
		endif
		if LocalCOB_Typ_481.bReserve4 = 1 then
			LocalCAN2Data.T1_By1 = BIT_SET(LocalCAN2Data.T1_By1, 7)
		else
			LocalCAN2Data.T1_By1 = BIT_CLR(LocalCAN2Data.T1_By1, 7)
		endif
; udPostennummer
			udShr16 = shr(LocalCOB_Typ_481.udPostennummer,16)
    	LocalCAN2Data.T1_By2_By3	= UINT(udShr16)							; take UPPERBytes of Prog/Kat ..
    	LocalCAN2Data.T1_By4_By5	= UINT(LocalCOB_Typ_481.udPostennummer)	; take LOWER byte..
; uiGewicht
		LocalCAN2Data.T1_By6_By7 = LocalCOB_Typ_481.uiGewicht

;****ID 481****Telegram 2********ID 481****Telegram 2********ID 481****Telegram 2********ID 481****Telegram 2****
;T2 mandatotries ->:
		LocalCAN2Data.T2_By0 		= BIT_SET(LocalCAN2Data.T2_By0, 5)
		LocalCAN2Data.T2_By0 		= BIT_CLR(LocalCAN2Data.T2_By0, 6)
		; .. and sign CAN2 telegram
		LocalCAN2Data.T2_By0 		= BIT_SET(LocalCAN2Data.T2_By0, 7)

; bProgKat
		if LocalCOB_Typ_481.bProgKat = 1 then
			LocalCAN2Data.T2_By0 = BIT_SET(LocalCAN2Data.T2_By0, 0)
		else
			LocalCAN2Data.T2_By0 = BIT_CLR(LocalCAN2Data.T2_By0, 0)
		endif

; Redundanzen -> T2-By0 - bit1..5
		if LocalCOB_Typ_481.bReserve5 = 1 then
			LocalCAN2Data.T2_By0 = BIT_SET(LocalCAN2Data.T2_By0, 1)
		else
			LocalCAN2Data.T2_By0 = BIT_CLR(LocalCAN2Data.T2_By0, 1)
		endif
		if LocalCOB_Typ_481.bReserve6 = 1 then
			LocalCAN2Data.T2_By0 = BIT_SET(LocalCAN2Data.T2_By0, 2)
		else
			LocalCAN2Data.T2_By0 = BIT_CLR(LocalCAN2Data.T2_By0, 2)
		endif
		if LocalCOB_Typ_481.bReserve7 = 1 then
			LocalCAN2Data.T2_By0 = BIT_SET(LocalCAN2Data.T2_By0, 3)
		else
			LocalCAN2Data.T2_By0 = BIT_CLR(LocalCAN2Data.T2_By0, 3)
		endif
		if LocalCOB_Typ_481.bReserve8 = 1 then
			LocalCAN2Data.T2_By0 = BIT_SET(LocalCAN2Data.T2_By0, 4)
		else
			LocalCAN2Data.T2_By0 = BIT_CLR(LocalCAN2Data.T2_By0, 4)
		endif
; Redundanzen..
		LocalCAN2Data.T2_By1 = LocalCOB_Typ_481.usReserve1
; uiProgKat
		LocalCAN2Data.T2_By2_By3 = LocalCOB_Typ_481.uiProgKat
; udKundennummer
			udShr16 = shr(LocalCOB_Typ_481.udKundennummer,16)
    	LocalCAN2Data.T2_By4_By5	= UINT(udShr16)							; take UPPERBytes of Prog/Kat ..
    	LocalCAN2Data.T2_By6_By7	= UINT(LocalCOB_Typ_481.udKundennummer)	; take LOWER byte..

;****ID 481****Telegram 3********ID 481****Telegram 3********ID 481****Telegram 3********ID 481****Telegramm 3****
;T2 mandatotries ->:
	LocalCAN2Data.T3_By0 		= BIT_CLR(LocalCAN2Data.T3_By0, 5)
	LocalCAN2Data.T3_By0 		= BIT_SET(LocalCAN2Data.T3_By0, 6)
	; .. and sign CAN2 telegram
	LocalCAN2Data.T3_By0 		= BIT_SET(LocalCAN2Data.T3_By0, 7)

	; Redundanzen
		if LocalCOB_Typ_481.bReserve9 = 1 then
			LocalCAN2Data.T3_By0 = BIT_SET(LocalCAN2Data.T3_By0, 1)
		else
			LocalCAN2Data.T3_By0 = BIT_CLR(LocalCAN2Data.T3_By0, 1)
		endif
		if LocalCOB_Typ_481.bReserve10 = 1 then
			LocalCAN2Data.T3_By0 = BIT_SET(LocalCAN2Data.T3_By0, 2)
		else
			LocalCAN2Data.T3_By0 = BIT_CLR(LocalCAN2Data.T3_By0, 2)
		endif

		; ###HO - 260905 - a_usCustomize[0..6]
		if(TARGETInfo_0.DataFormat = 2) then  ; motorola
			memcpy(adr(LocalCAN2Data.T3_By1),adr(LocalCOB_Typ_481.a_usCustomize[0]),1)
			memcpy(adr(LocalCAN2Data.T3_By2_By3),adr(LocalCOB_Typ_481.a_usCustomize[1]),2)
			memcpy(adr(LocalCAN2Data.T3_By4_By5),adr(LocalCOB_Typ_481.a_usCustomize[3]),2)
			memcpy(adr(LocalCAN2Data.T3_By6_By7),adr(LocalCOB_Typ_481.a_usCustomize[5]),2)
		else ; intel
			LocalCAN2Data.T3_By1	 = LocalCOB_Typ_481.a_usCustomize[0]
			LocalCAN2Data.T3_By2_By3 = LocalCOB_Typ_481.a_usCustomize[2] + 256* LocalCOB_Typ_481.a_usCustomize[1]
			LocalCAN2Data.T3_By4_By5 = LocalCOB_Typ_481.a_usCustomize[4] + 256* LocalCOB_Typ_481.a_usCustomize[3]
			LocalCAN2Data.T3_By6_By7 = LocalCOB_Typ_481.a_usCustomize[6] + 256* LocalCOB_Typ_481.a_usCustomize[5]
		endif

     iStatus = 0
     pCAN2Data = ADR(LocalCAN2Data)
endaction ; ID 481

; *** add new COBs here.. ***

; the other IDs that have not been defined below that are not supported by this Lib..
elseaction:
    	iStatus = 110
endaction

endcase

ENDE:
;********************************************************************************************************
;********************************************************************************************************

;********************************************************************************************************
;********************************************************************************************************
; use to add new COB .. ->
;********************************************************************************************************
;********************************************************************************************************

;*******action xxx********action xxx********action xxx********action xxx********action xxx********
(*

action xxx:
	    ; to do: transform LocalHFAnWaschm_ObjNr120_type data to LocalCAN2Data
  		memcpy(adr(LocalCOB_Typ_xxx),Local_InitCAN2PV.pPVData,sizeof(LocalCOB_Typ_xxx))

;****ID xxx****Telegram 1********ID xxx****Telegram 1********ID xxx****Telegram 1********ID xxx****Telegram 1****
;T1 mandatotries ->:
		LocalCAN2Data.T1_By0 = BIT_CLR(LocalCAN2Data.T1_By0, 5)
		LocalCAN2Data.T1_By0 = BIT_CLR(LocalCAN2Data.T1_By0, 6)
		; .. and sign CAN2 telegram
		LocalCAN2Data.T1_By0 = BIT_SET(LocalCAN2Data.T1_By0, 7)
;BOOL->:
		; bBereit
    	if pLocalHFAnWaschm_ObjNr120.bBereit = 1 then
			LocalCAN2Data.T1_By0 = BIT_SET(LocalCAN2Data.T1_By0, 0)
		else
			LocalCAN2Data.T1_By0 = BIT_CLR(LocalCAN2Data.T1_By0, 0)
		endif
;USINT->:
		; usFehlernummer
		LocalCAN2Data.T1_By1 	= pLocalHFAnWaschm_ObjNr120.usFehlernummer
;UDINT->:
		; broadcast via CAN in 'motorola order' : MSByte as byte2 and LSByte as byte5 !!
			udShr16 = shr(pLocalHFAnWaschm_ObjNr120.udPostennummer	,16)
    	LocalCAN2Data.T1_By2_By3	= UINT(udShr16)										; take UPPERBytes of Prog/Kat ..
    	LocalCAN2Data.T1_By4_By5	= UINT(pLocalHFAnWaschm_ObjNr120.udPostennummer)	; take LOWER byte..
;UINT->
		; uiGewicht
    	LocalCAN2Data.T1_By6_By7	= pLocalHFAnWaschm_ObjNr120.uiGewicht

;****ID xxx****Telegram 2********ID xxx****Telegram 2********ID xxx****Telegram 2********ID xxx****Telegram 2****
;T2 mandatotries ->:
		LocalCAN2Data.T2_By0					= BIT_SET(LocalCAN2Data.T2_By0, 5)
		LocalCAN2Data.T2_By0  					= BIT_CLR(LocalCAN2Data.T2_By0, 6)
		; .. and sign CAN2 telegram
		LocalCAN2Data.T2_By0 					= BIT_SET(LocalCAN2Data.T2_By0, 7)
		LocalCAN2Data.T1_By0 = BIT_SET(LocalCAN2Data.T1_By0, 7)
;BOOL->:
		; bProgrammOderKategorie
    	if pLocalHFAnWaschm_ObjNr120.bProgrammOderKategorie = 1 then
			LocalCAN2Data.T2_By0 				= BIT_SET(LocalCAN2Data.T2_By0, 0)
		else
			LocalCAN2Data.T2_By0 				= BIT_CLR(LocalCAN2Data.T2_By0, 0)
		endif
;UINT->
		; uiProgrammKategorie
    	LocalCAN2Data.T2_By2_By3	= pLocalHFAnWaschm_ObjNr120.uiProgrammKategorie
;UDINT->:
	   	; udKundennummer
	   		udShr16 = shr(pLocalHFAnWaschm_ObjNr120.udKundennummer	,16)
		; broadcast via can in motorola format: MSByte as byteN and LSByte as byteN+1 !!
    	LocalCAN2Data.T2_By4_By5	= UINT(udShr16)								; take UPPERBytes of Prog/Kat ..
    	LocalCAN2Data.T2_By6_By7	= UINT(pLocalHFAnWaschm_ObjNr120.udKundennummer	)	; take LOWER byte..

;****ID xxx****Telegram 3********ID xxx****Telegram 3********ID xxx****Telegram 3********ID xxx****Telegram 3****
;T3 mandatotries ->:
		LocalCAN2Data.T3_By0					= BIT_CLR(LocalCAN2Data.T3_By0, 5)
		LocalCAN2Data.T3_By0 					= BIT_SET(LocalCAN2Data.T3_By0, 6)
		; .. and sign CAN2 telegram
		LocalCAN2Data.T3_By0 					= BIT_SET(LocalCAN2Data.T3_By0, 7)
;AKZ as STRING->:
		; "Auftragskennzeichen" as string has to be set to T3 + T4..
		; always assure transmitting this order:
		; T3Byte2 -> zchn1 ; T4Byte7 -> zchn 12 (quasi-motorola order)

		pLocByte4Str access (Local_InitCAN2PV.adr_data + 14) ; don't use static address !!!
		LocByte4Str = pLocByte4Str

		LocalCAN2Data.T3_By2_By3	= UINT(pLocByte4Str[0])
		LocalCAN2Data.T3_By2_By3	= shl(LocalCAN2Data.T3_By2_By3, 8)
		LocalCAN2Data.T3_By2_By3	= LocalCAN2Data.T3_By2_By3 + pLocByte4Str[1]

		LocalCAN2Data.T3_By4_By5	= UINT(pLocByte4Str[2])
		LocalCAN2Data.T3_By4_By5	= shl(LocalCAN2Data.T3_By4_By5, 8)
		LocalCAN2Data.T3_By4_By5	= LocalCAN2Data.T3_By4_By5 + pLocByte4Str[3]

		LocalCAN2Data.T3_By6_By7	= UINT(pLocByte4Str[4])
		LocalCAN2Data.T3_By6_By7	= shl(LocalCAN2Data.T3_By6_By7, 8)
		LocalCAN2Data.T3_By6_By7	= LocalCAN2Data.T3_By6_By7 + pLocByte4Str[5]

;****ID xxx****Telegram 4********ID xxx****Telegram 4********ID xxx****Telegram 4********ID xxx****Telegram 4****
;T3 mandatotries ->:
		LocalCAN2Data.T4_By0 				= BIT_SET(LocalCAN2Data.T4_By0, 5)
		LocalCAN2Data.T4_By0 				= BIT_SET(LocalCAN2Data.T4_By0, 6)
		; .. and sign CAN2 telegram
		LocalCAN2Data.T4_By0 = BIT_SET(LocalCAN2Data.T4_By0, 7)
;AKZ as STRING->:
		LocalCAN2Data.T4_By2_By3	= UINT(pLocByte4Str[6])
		LocalCAN2Data.T4_By2_By3	= shl(LocalCAN2Data.T4_By2_By3, 8)
		LocalCAN2Data.T4_By2_By3	= LocalCAN2Data.T4_By2_By3 + pLocByte4Str[7]

		LocalCAN2Data.T4_By4_By5	= UINT(pLocByte4Str[8])
		LocalCAN2Data.T4_By4_By5	= shl(LocalCAN2Data.T4_By4_By5, 8)
		LocalCAN2Data.T4_By4_By5	= LocalCAN2Data.T4_By4_By5 + pLocByte4Str[9]

		LocalCAN2Data.T4_By6_By7	= UINT(pLocByte4Str[10])
		LocalCAN2Data.T4_By6_By7	= shl(LocalCAN2Data.T4_By6_By7, 8)
		LocalCAN2Data.T4_By6_By7	= LocalCAN2Data.T4_By6_By7 + pLocByte4Str[11]

        iStatus = 0
        pCAN2Data = ADR(LocalCAN2Data)

endaction ; ID xxx
*)

;********************************************************************************************************
;********************************************************************************************************

	; check swapping and casting..
(*	x 	= $89abcdef			; -> 16# 89 ab cd ef
	xswap 	= swapUDINT(x)	; -> 16# ef cd ab 89
	uiCastx = UINT(x)		; -> 16# cd ef
	udSHR4x = shr(x,16)		; -> 16# 00 00 89 ab *)

;********************************************************************************************************
;********************************************************************************************************

END_FUNCTION_BLOCK
```

#### CAN2RW.ab
```automation-basic
FUNCTION_BLOCK CAN2RW
;********************************************************************************************************
; * Implementation of CAN2RW
;********************************************************************************************************
; * version 		3.2.1
; * last change		111007
; * by				H.O.
;********************************************************************************************************
; * history:
;***********
; V3.2.1 - ###hcs/HO - 101007
; 	COB_ID130und140 und COB_ID131und141 entfernt - stattdessen Neudefinition:
; 		* COB 130 und COB140 wie COB120
;		* COB131 und COB141 wie COB121
; 	* V2.0.0:
;		* InPara 'p_InitCAN2Protocol' replaced by DO 'AdrIC2Prot'
; 		* Communication-globalPara 'CAN2Init.iMode' replaced by COB-individual-parameter 'InitCAN2PV.iMode'
; 		* mode by that telegrams have been sent within cycletime changed:
;		* 200ms - exclusively between tels with identical CANID
; 		* all tels of WETCAN2Tel are sent immediately
; 	* V2.1.0
;		* DO "AdrIC2Prot" replaced by pCAN2Init_ident
; 		* enable added
; 	* V3.1.0 - 141206 ###HO
;		* COB126+128 bei COB120 verodert
;********************************************************************************************************
;********************************************************************************************************

if (enable = 0) then
	goto ENDE
endif

uiStatusEvVar 	= 105 ; never return 105..
uiStatus		= 105
;***************************************************************************
; check for target platform - motorola or intel ..
TARGETInfo_0.enable		= 1
TARGETInfo_0.pOSVersion	= ADR(pOSVersion)
TARGETInfo_0 FUB TARGETInfo()

if(TARGETInfo_0.DataFormat = 1) then
	bIntel 		= TRUE
	bMotorola 	= FALSE
else
	bIntel 		= FALSE
	bMotorola 	= TRUE
endif
;***************************************************************************
; as no pointer has been passed in - get ID of AdressDO again..
; ###HO 080404 handle reactivated..
p_InitCAN2Protocol = pCAN2Init_ident
(*
DatObjInfo(1, "AdrIC2Prot", DO_StatInfo, DO_IDAdrInitCan2Prot, DO_StartAdr, DO_Len, DO_Memtype, DO_Option, DO_ChangeDat )
; get address for initdata..
DatObjRead_AdrIC2Prot.enable			= 1
DatObjRead_AdrIC2Prot.ident			= DO_IDAdrInitCan2Prot
DatObjRead_AdrIC2Prot.Offset			= 0
DatObjRead_AdrIC2Prot.pDestination	= adr(p_InitCAN2Protocol)
DatObjRead_AdrIC2Prot.len			= 4
DatObjRead_AdrIC2Prot FUB DatObjRead()
*)
; get local structure with initdata..
memcpy(adr(Local_InitCAN2Protocol),p_InitCAN2Protocol,sizeof(Local_InitCAN2Protocol))

;***************************************************************************
; prepare reading from InitDO (type '_InitCAN2PV' )..
DatObjRead_fromInitDO.enable	= 1 												; enable is always "1"
DatObjRead_fromInitDO.ident		= Local_InitCAN2Protocol.AccessInitDO.DO_us_ident 	; user ID of DO..
DatObjRead_fromInitDO.len		= sizeof(Local_InitCAN2PV)  						; size of a single data record..

; prepare reading from DORead..
DatObjRead_fromDORead.enable 	= 1
DatObjRead_fromDORead.ident		= Local_InitCAN2Protocol.DOAccessCAN2Read.DO_us_ident

; prepare writing to DORead..
DatObjWrite_toDORead.enable		= 1
DatObjWrite_toDORead.ident		= Local_InitCAN2Protocol.DOAccessCAN2Read.DO_us_ident

; prepare reading from DOWrite..
DatObjRead_fromDOWrite.enable	= 1
DatObjRead_fromDOWrite.ident	= Local_InitCAN2Protocol.DoAccessCAN2Write.DO_us_ident

; prepare writing to DOWrite..
DatObjWrite_toDOWrite.enable	= 1
DatObjWrite_toDOWrite.ident		= Local_InitCAN2Protocol.DoAccessCAN2Write.DO_us_ident
;***************************************************************************

loop iLoopIdx = 0 to (Local_InitCAN2Protocol.CAN2DObCount -1) do
	; get COB specific data from InitDO..
	DatObjRead_fromInitDO.Offset		= iLoopIdx * sizeof(Local_InitCAN2PV)
	DatObjRead_fromInitDO.len			= sizeof(Local_InitCAN2PV)
	DatObjRead_fromInitDO.pDestination	= adr(Local_InitCAN2PV)
	DatObjRead_fromInitDO FUB DatObjRead()
	if(uiStatus = 105) then
		uiStatus = DatObjRead_fromInitDO.status
	endif
;---write---write---write---write---write---write---write---write---write---write---write---write
	if(Local_InitCAN2PV.usCommDirection) = 1 then 	; write COB
		; read from DOWrite to decide if write operation is necessary ..
		; read from DO -> necessary to get time when last tel has been sent..
		DatObjRead_fromDOWrite.Offset		= iLoopIdx * sizeof(LocalCAN2Write)
		DatObjRead_fromDOWrite.len			= sizeof(LocalCAN2Write)
		DatObjRead_fromDOWrite.pDestination	= adr(LocalCAN2Write)
		DatObjRead_fromDOWrite FUB DatObjRead()
		if(uiStatus = 0) then
			uiStatus = DatObjRead_fromDOWrite.status
		endif
;---write-auto mode---write-auto mode--- write-auto modewrite-auto mode---write-auto mode---

		; V2.0.0 -> Local_InitCAN2Protocol.iMode replaced by Local_InitCAN2PV.iMode..
		if(Local_InitCAN2PV.iMode = 0 ) then ; '0' -> cyclic mode

			tActTime = GetTime()
			tDiffTime = DiffT(tActTime, LocalCAN2Write.tTimeLastTelSent)
			if ( tDiffTime > 187 ) then ; 200ms has been elapsed..
				; read PV..
				_SetCAN2COBTypeToCAN2Type_0.p_InitCAN2PV = adr(Local_InitCAN2PV)
				_SetCAN2COBTypeToCAN2Type_0 FUB _SetCAN2COBTypeToCAN2Type()
				; now - LocalCAN2Copy contains data to send..
				memcpy (adr(LocalCAN2Copy), _SetCAN2COBTypeToCAN2Type_0.pCAN2Data, sizeof(LocalCAN2Copy))

				_GetCANIDFromObjNr_0.udObjNr =  UDINT(Local_InitCAN2PV.uiObjNr)
				_GetCANIDFromObjNr_0 FUB _GetCANIDFromObjNr()

				; ###HO - 110205 - Steuerung #Tels zur Laufzeit (bislang in Init festgelegt !)
				; (!) (hierein gehören eigentlich keine COB-spezifischen Dinge)
				iTempNumberOfTels = 0
				;###HO -141206 126,128 added..
				if ((Local_InitCAN2PV.uiObjNr = 120)or(Local_InitCAN2PV.uiObjNr = 126)or(Local_InitCAN2PV.uiObjNr = 128)\
					or(Local_InitCAN2PV.uiObjNr = 130)or(Local_InitCAN2PV.uiObjNr = 140)) then ;###HO 111007
					if Bit_Tst (LocalCAN2Copy.T1_By0,3) then ; #tels =4
						iTempNumberOfTels = 5
					else ; #tels= 2
						iTempNumberOfTels = 3
					endif
				else
					iTempNumberOfTels = LocalCAN2Write.iNumberOfTels
				endif

				loop iTelsSendIdx = 1 to iTempNumberOfTels do
					; send 1st telegram now..

					CANquwr_1.enable	= 1
					CANquwr_1.us_ident	= Local_InitCAN2Protocol.CANAccess.CANopen_us_ident
					CANquwr_1.can_id	= _GetCANIDFromObjNr_0.udObjNr
					if (bMotorola = TRUE) then
						_SetCAN2TypeToCAN1Type_0.pCAN2Data		= adr(LocalCAN2Copy)
						_SetCAN2TypeToCAN1Type_0.iTelegramIndex	= iTelsSendIdx
						_SetCAN2TypeToCAN1Type_0 FUB _SetCAN2TypeToCAN1Type()
						CANquwr_1.data_adr	= _SetCAN2TypeToCAN1Type_0.pCAN1Data
					else if (bIntel = TRUE) then
						_Seti386CAN2TypeToCAN1Type_0.pCAN2Data		= adr(LocalCAN2Copy)
						_Seti386CAN2TypeToCAN1Type_0.iTelegramIndex	= iTelsSendIdx
						_Seti386CAN2TypeToCAN1Type_0 FUB _Seti386CAN2TypeToCAN1Type()
						CANquwr_1.data_adr	= _Seti386CAN2TypeToCAN1Type_0.pCAN1Data
					else
						uiStatus = TARGETInfo_0.status
					endif
					CANquwr_1.data_lng	= 8
					CANquwr_1 FUB CANquwr()
					if(CANquwr_1.status = 0) then 	; sending tel succeeded
						LocalCAN2Write.tTimeLastTelSent = GetTime()
					else 							; sending tel failed
						LocalCAN2Write.tTimeLastTelSent = TIME(0)
					endif 							; CANquwr_1.status = 0 ?
				endloop
				; return last status of CANquwr() to EvVar..
				uiStatusEvVar = CANquwr_1.status
				memcpy(Local_InitCAN2PV.pEvVar,adr(uiStatusEvVar), sizeof(uiStatusEvVar))
			else	; 200ms has not been elapsed yet..
				; do nothing -> wait..
			endif

;---write-EvControlled---write-EvControlled--- write-EvControlledwrite-EvControlled---write-EvControlled---

		; V2.0.0 -> Local_InitCAN2Protocol.iMode replaced by Local_InitCAN2PV.iMode
		else if (Local_InitCAN2PV.iMode = 1) then ; '1' -> manually mode
				; always check EvVar to decide about WriteOperation..
				memcpy (adr(uiLocalEvVar),Local_InitCAN2PV.pEvVar,sizeof(uiLocalEvVar))
				if(uiLocalEvVar = 1) then ; user defines writing to CAN..

					tActTime = GetTime()
					tDiffTime = DiffT(tActTime, LocalCAN2Write.tTimeLastTelSent)
					if ( tDiffTime > 187 ) then ; 200ms has been elapsed..
						; expected behavior ? process image should be read whether user decides - save and send if time expired..
						; read PV..
						_SetCAN2COBTypeToCAN2Type_0.p_InitCAN2PV = adr(Local_InitCAN2PV)
						_SetCAN2COBTypeToCAN2Type_0 FUB _SetCAN2COBTypeToCAN2Type()
						; now - LocalCAN2Copy contains data to send..
						memcpy (adr(LocalCAN2Copy), _SetCAN2COBTypeToCAN2Type_0.pCAN2Data, sizeof(LocalCAN2Copy))

						_GetCANIDFromObjNr_0.udObjNr =  UDINT(Local_InitCAN2PV.uiObjNr)
						_GetCANIDFromObjNr_0 FUB _GetCANIDFromObjNr()

						; ###HO - 110205 - Steuerung #Tels zur Laufzeit (bislang in Init festgelegt !)
						; (!) (hierein gehören eigentlich keine COB-spezifischen Dinge)
						iTempNumberOfTels = 0
						if ((Local_InitCAN2PV.uiObjNr = 120)or(Local_InitCAN2PV.uiObjNr = 126)or(Local_InitCAN2PV.uiObjNr = 128)\
							or(Local_InitCAN2PV.uiObjNr = 130)or(Local_InitCAN2PV.uiObjNr = 140)) then ;###HO -111007
							if Bit_Tst (LocalCAN2Copy.T1_By0,3) then ; #tels =4
								iTempNumberOfTels = 5
							else ; #tels= 2
								iTempNumberOfTels = 3
							endif
						else
							iTempNumberOfTels = LocalCAN2Write.iNumberOfTels
						endif

						loop iTelsSendIdx = 1 to iTempNumberOfTels do ;LocalCAN2Write.iNumberOfTels
							; send 1st telegram now..

							CANquwr_1.enable	= 1
							CANquwr_1.us_ident	= Local_InitCAN2Protocol.CANAccess.CANopen_us_ident
							CANquwr_1.can_id	= _GetCANIDFromObjNr_0.udObjNr
							if (bMotorola = TRUE) then
								_SetCAN2TypeToCAN1Type_0.pCAN2Data		= adr(LocalCAN2Copy)
								_SetCAN2TypeToCAN1Type_0.iTelegramIndex	= iTelsSendIdx
								_SetCAN2TypeToCAN1Type_0 FUB _SetCAN2TypeToCAN1Type()
								CANquwr_1.data_adr	= _SetCAN2TypeToCAN1Type_0.pCAN1Data
							else if (bIntel = TRUE) then
								_Seti386CAN2TypeToCAN1Type_0.pCAN2Data		= adr(LocalCAN2Copy)
								_Seti386CAN2TypeToCAN1Type_0.iTelegramIndex	= iTelsSendIdx
								_Seti386CAN2TypeToCAN1Type_0 FUB _Seti386CAN2TypeToCAN1Type()
								CANquwr_1.data_adr	= _Seti386CAN2TypeToCAN1Type_0.pCAN1Data
							else
								uiStatus = TARGETInfo_0.status
							endif
							CANquwr_1.data_lng	= 8
							CANquwr_1 FUB CANquwr()
							if(CANquwr_1.status = 0) then 	; sending tel succeeded
								LocalCAN2Write.tTimeLastTelSent = GetTime()
							else 							; sending tel failed
								LocalCAN2Write.tTimeLastTelSent = TIME(0)
							endif 							; CANquwr_1.status = 0 ?
						endloop
						; return last status of CANquwr() to EvVar..
						uiStatusEvVar = CANquwr_1.status
						memcpy(Local_InitCAN2PV.pEvVar,adr(uiStatusEvVar), sizeof(uiStatusEvVar))

					else	; 200ms has not been elapsed yet..
						; do nothing -> wait..
					endif
				else ; EvVar <> 'WriteNow!'
					; do nothing -> wait and goto next COB..
				endif	; EvVar defined as 'WriteNow!'
			endif

;***********read operation*************	read operation*************read operation*****************

	else if(Local_InitCAN2PV.usCommDirection) = 0 then	; read COB ,
;---read-EvControlled---read-EvControlled--- read-EvControlledread-EvControlled---read-EvControlled---

		; V2.0.0 -> Local_InitCAN2Protocol.iMode replaced by Local_InitCAN2PV.iMode
		if(Local_InitCAN2PV.iMode = 1 ) then ; '1' -> manually mode
			; to do read operation.. auto mode/man mode: same procedure as..

			; for new COB -> delete LocalCAN1Data
			LocalCAN1Data.T_By0 	= 0
			LocalCAN1Data.T_By1 	= 0
			LocalCAN1Data.T_By2_By3 = 0
			LocalCAN1Data.T_By4_By5 = 0
			LocalCAN1Data.T_By6_By7 = 0

			bOverwritePV = FALSE

			; reset local CAN2 buffer before reding from queue..
			loop iIdx = 0 to 49 do		; ###HO - 02.09.2005
				LocalCAN2Read.ab_ByteArray[iIdx] 	= 0
				LocalCAN2ReadBak.ab_ByteArray[iIdx] = 0
			endloop

			memcpy (adr(uiLocalEvVar),Local_InitCAN2PV.pEvVar,sizeof(uiLocalEvVar))
			if (uiLocalEvVar = 1 ) then ; uiLocalEvVar = 1 -> user decided to read from queue

				loop	; check queue for received telegrams and reassemble them..

					CANrd_0.enable		= 1
					CANrd_0.q_ident		= Local_InitCAN2PV.udCAN_q_ident
					CANrd_0.data_adr	= ADR(LocalCAN1Data)
					CANrd_0 FUB CANrd()

					if(CANrd_0.status = 0) then ; CAN tel found in queue .. ; CANrd_0.status == 0 ?
						; one tel could be read successfully -> reading from queue is running..

						; set actual tel to can2 struct
						_GetCANIDFromObjNr_0.udObjNr	= UDINT(Local_InitCAN2PV.uiObjNr)
						_GetCANIDFromObjNr_0 FUB _GetCANIDFromObjNr()

						_SetCAN1TypeToByteArray_0.a_usInByteArray	= LocalCAN2Read.ab_ByteArray
						_SetCAN1TypeToByteArray_0.udCanID			= _GetCANIDFromObjNr_0.udCANID
						_SetCAN1TypeToByteArray_0.CAN1Data			= LocalCAN1Data
						_SetCAN1TypeToByteArray_0 FUB _SetCAN1TypeToByteArray()

						; save OutArray to local array - in dependency of target platform
	 					LocalCAN2Read.ab_ByteArray = _SetCAN1TypeToByteArray_0.a_usOutByteArray
						; dont convert platform dependent ! convert when overwrite PV !

						uiStatusEvVar = 710
						memcpy(Local_InitCAN2PV.pEvVar,adr(uiStatusEvVar), sizeof(uiStatusEvVar))

						if(_SetCAN1TypeToByteArray_0.bDataValid = TRUE ) then ;_SetCAN1TypeToByteArray_0.bDataValid == TRUE ?
							LocalCAN2ReadBak.ab_ByteArray = LocalCAN2Read.ab_ByteArray
							bOverwritePV = TRUE

						else 	;_SetCAN1TypeToByteArray_0.bDataValid == TRUE ?
							; do nothing - continue reading from queue..
						endif	;_SetCAN1TypeToByteArray_0.bDataValid == TRUE ?

					else if(CANrd_0.status = 8877) then  	; CANrd_0.status == 0 ?
							if(bOverwritePV = TRUE )then  ; bOverwritePV == TRUE ?
								; complete CAN2 tel has been found in queue - return '1' to EvVar..
								uiStatusEvVar = 0
								memcpy(Local_InitCAN2PV.pEvVar,adr(uiStatusEvVar), sizeof(uiStatusEvVar))

								loop iResIdx = 0 to 49 do ;###HO -020905
									ab_ByteArrayi386Temp[iResIdx] = 0
								endloop

								; now- it's time to overwrite PV
								_GetPVSize_0.uiObjNr = Local_InitCAN2PV.uiObjNr
								_GetPVSize_0 FUB _GetPVSize()

								if (bMotorola = TRUE) then
									ab_ByteArrayi386Temp = LocalCAN2ReadBak.ab_ByteArray
								else if (bIntel = TRUE) then
									_ConvertDataToi386_1.uiObjNr			= Local_InitCAN2PV.uiObjNr
									_ConvertDataToi386_1.ByteArrayMotorola	= LocalCAN2ReadBak.ab_ByteArray
									_ConvertDataToi386_1 FUB _ConvertDataToi386()

									ab_ByteArrayi386Temp = _ConvertDataToi386_1.ByteArrayi386

									else
										uiStatus = TARGETInfo_0.status
									endif

							 	memcpy(	Local_InitCAN2PV.pPVData, adr(ab_ByteArrayi386Temp), _GetPVSize_0.iCobLength)
							 										; LocalCAN2ReadBak.ab_ByteArray
								bOverwritePV = FALSE

								; exit loop..
								exitif (TRUE = TRUE)
							else	; bOverwritePV == TRUE ?
								; return errcode - less tels as necessary for complete CAN2 tel has been found in queue..
								uiStatusEvVar = 8877
								memcpy(Local_InitCAN2PV.pEvVar,adr(uiStatusEvVar), sizeof(uiStatusEvVar))

								; exit loop..
								exitif (TRUE = TRUE)
							endif	; bOverwritePV == TRUE ?

					else ; CANrd_0.status neither 0 nor 8877
						uiStatusEvVar = CANrd_0.status
						memcpy(Local_InitCAN2PV.pEvVar,adr(uiStatusEvVar), sizeof(uiStatusEvVar))

						; exit loop..
						exitif (TRUE = TRUE)
					endif	; CANrd_0.status == 0 ?

				endloop	; reading whole queue..

			else ; all other states of EvVar except '1'
				; do nothing..
			endif ; uiLocalEvVar == 1 ?,

;---read-auto mode---read-auto mode--- read-EvControlledread-auto mode---read-auto mode---

		; V2.0.0 -> Local_InitCAN2Protocol.iMode replaced by Local_InitCAN2PV.iMode ..
		else if (Local_InitCAN2PV.iMode = 0) then	 ; auto mode
		; be aware: reading in auto mode is faster than tels have to be set in queue by write operation..
		; -> use DORead..
			; for new COB -> delete LocalCAN1Data
			LocalCAN1Data.T_By0 	= 0
			LocalCAN1Data.T_By1 	= 0
			LocalCAN1Data.T_By2_By3 = 0
			LocalCAN1Data.T_By4_By5 = 0
			LocalCAN1Data.T_By6_By7 = 0

			bOverwritePV = FALSE

			; reset local CAN2 buffer before reding from queue..
			loop iIdx = 0 to 49 do	; ###HO - 020905
				LocalCAN2Read.ab_ByteArray[iIdx] 	= 0
				LocalCAN2ReadBak.ab_ByteArray[iIdx] = 0
			endloop

			loop	; check queue for received telegrams and reassemble them..

				CANrd_0.enable		= 1
				CANrd_0.q_ident		= Local_InitCAN2PV.udCAN_q_ident
				CANrd_0.data_adr	= ADR(LocalCAN1Data)
				CANrd_0 FUB CANrd()

				if(CANrd_0.status = 0) then ; CAN tel found in queue .. ; CANrd_0.status == 0 ?
					; one tel could be read successfully -> reading from queue is running..

					DatObjRead_fromDORead.enable 		= 1
					DatObjRead_fromDORead.ident			= Local_InitCAN2Protocol.DOAccessCAN2Read.DO_us_ident
					DatObjRead_fromDORead.Offset		= iLoopIdx * sizeof(LocalCAN2Read)
					DatObjRead_fromDORead.pDestination	= adr(LocalCAN2Read)
					DatObjRead_fromDORead.len			= sizeof(LocalCAN2Read)
					DatObjRead_fromDORead FUB DatObjRead()

					; set actual tel to can2 struct
					_GetCANIDFromObjNr_0.udObjNr	= UDINT(Local_InitCAN2PV.uiObjNr)
					_GetCANIDFromObjNr_0 FUB _GetCANIDFromObjNr()

					_SetCAN1TypeToByteArray_0.a_usInByteArray	= LocalCAN2Read.ab_ByteArray
					_SetCAN1TypeToByteArray_0.udCanID			= _GetCANIDFromObjNr_0.udCANID
					_SetCAN1TypeToByteArray_0.CAN1Data			= LocalCAN1Data
					_SetCAN1TypeToByteArray_0 FUB _SetCAN1TypeToByteArray()

					LocalCAN2Read.ab_ByteArray = _SetCAN1TypeToByteArray_0.a_usOutByteArray

					; status 'running' doesn't match -> why ?

					; last telegram has been read ?
					if(_SetCAN1TypeToByteArray_0.bDataValid = TRUE ) then ;_SetCAN1TypeToByteArray_0.bDataValid == TRUE ?
						LocalCAN2ReadBak.ab_ByteArray = LocalCAN2Read.ab_ByteArray
						bOverwritePV = TRUE

						; reset buffer to write back to DORead..
						loop iIdx = 0 to 49 do
							LocalCAN2Read.ab_ByteArray[iIdx] 	= 0
						endloop

					else 	;_SetCAN1TypeToByteArray_0.bDataValid == TRUE ?
						; do nothing - continue reading from queue..
					endif	;_SetCAN1TypeToByteArray_0.bDataValid == TRUE ?

					; tel has been read successfully -> set to DORead
					DatObjWrite_toDORead.Offset		= iLoopIdx * sizeof(LocalCAN2Read)
					DatObjWrite_toDORead.pSource	= adr(LocalCAN2Read)
					DatObjWrite_toDORead.len		= sizeof(LocalCAN2Read)
					DatObjWrite_toDORead FUB DatObjWrite()

				else if(CANrd_0.status = 8877) then  	; CANrd_0.status == 0 ?
						if(bOverwritePV = TRUE )then  ; bOverwritePV == TRUE ?
							; complete CAN2 tel has been found in queue - return '1' to EvVar..
							uiStatusEvVar = 0
							memcpy(Local_InitCAN2PV.pEvVar,adr(uiStatusEvVar), sizeof(uiStatusEvVar))

							loop iResIdx = 0 to 49 do ;###HO -020905
								ab_ByteArrayi386Temp[iResIdx] = 0
							endloop

							; now- it's time to overwrite PV
							_GetPVSize_0.uiObjNr = Local_InitCAN2PV.uiObjNr
							_GetPVSize_0 FUB _GetPVSize()

							if (bMotorola = TRUE) then
								ab_ByteArrayi386Temp = LocalCAN2ReadBak.ab_ByteArray
							else if (bIntel = TRUE) then
								_ConvertDataToi386_1.uiObjNr			= Local_InitCAN2PV.uiObjNr
								_ConvertDataToi386_1.ByteArrayMotorola	= LocalCAN2ReadBak.ab_ByteArray
								_ConvertDataToi386_1 FUB _ConvertDataToi386()

								ab_ByteArrayi386Temp = _ConvertDataToi386_1.ByteArrayi386

								else
									uiStatus = TARGETInfo_0.status
							endif
						 	memcpy(	Local_InitCAN2PV.pPVData, adr(ab_ByteArrayi386Temp), _GetPVSize_0.iCobLength)

							bOverwritePV = FALSE

							; exit loop..
							exitif (TRUE = TRUE)
						else	; bOverwritePV == TRUE ?
							; return errcode - less tels as necessary for complete CAN2 tel has been found in queue..
							uiStatusEvVar = 8877
							memcpy(Local_InitCAN2PV.pEvVar,adr(uiStatusEvVar), sizeof(uiStatusEvVar))

							; exit loop..
							exitif (TRUE = TRUE)
						endif	; bOverwritePV == TRUE ?

				else ; CANrd_0.status neither 0 nor 8877
					uiStatusEvVar = CANrd_0.status
					memcpy(Local_InitCAN2PV.pEvVar,adr(uiStatusEvVar), sizeof(uiStatusEvVar))

					; exit loop..
					exitif (TRUE = TRUE)
				endif	; CANrd_0.status == 0 ?

			endloop	; reading whole queue..

		else	; iMode neither '0' nor '1'
			; uiStatus = 560
			; don't copy to EvVar -> this is a 'global problem'
			; -> from V2.0.0 -> no global problem any more..
			memcpy(Local_InitCAN2PV.pEvVar,adr(uiStatus),sizeof(uiStatus))
		endif
	else ; CommDirection neither 0 nor 1 passed by user
		uiStatus = 520
		; don't copy to EvVar -> this is a 'global problem'
		; memcpy(Local_InitCAN2PV.pEvVar,adr(uiStatus),sizeof(uiStatus))
	endif ; CommDirection 0 or 1 or error

	; always write back to DOWrite..
	DatObjWrite_toDOWrite.Offset		= iLoopIdx * sizeof(LocalCAN2Write)
	DatObjWrite_toDOWrite.pSource		= adr(LocalCAN2Write)
	DatObjWrite_toDOWrite.len			= sizeof(LocalCAN2Write)
	DatObjWrite_toDOWrite FUB DatObjWrite()

	if(uiStatus = 0) then
		uiStatus = DatObjWrite_toDOWrite.status
	endif

endloop ; reading all COBs..

;********************************************************************************************************
ENDE:
;********************************************************************************************************
END_FUNCTION_BLOCK
```
